(* IEC 61131-3 sources: std_i2980_v2.06_cp053/Source/IMM/ieccontrol/InjectionGeneral (part 8) *)

(* ---- ABInjectionCalibCycle.pu ---- *)
(*
@h    ! WARNING !
@h    The Kemro K2 system (including software) only meets category B according to EN 954-1,
@h    thus it is not intended for usage in safety-relevant control applications in the field
@h    of personal safety (e.g. emergency stop).
@h    To implement potentially necessary safety-relevant control tasks, always use additional
@h    external safety devices that are intended for the particular purpose, and meet the necessary
@h    functional safety.
@h    For further information see EN 954-1 (EN ISO 13849-1) and/or the K2-x00 user manual, chapter
@h    "CE conformity, directives and standards".

Do steps for automatic injection calibration (plant/dead time analysis)
*)

IMPORT_OVER_LISTFILE
 SET_EVENT
, SET_ALARM
, KMEM_ArrayCreate
, KMEM_ArraySet
, KMEM_ArrayDelete
, tnCalibMode_Both
, tnCalibState_Error
, tnCalibState_Aborted
, cMaxInjectionCount
, tnCalibMode_Raising
, tnCalibMode_Falling
, tnCalibState_Done
, cMoveFwd
, cMoveInject
, cMoveInjectCalib
, cMoveBwd
, cMoveDecompAftPlast
, nSetup
, tnCalibState_Running
, cCalibShiftData
, cCalibMeasuredVel
, cCalibMeasuredOutput
, tsControlParameters
, tnOperationMode
, tsDeviceId
, tsCalibMovement
, tsCalculatedInjectData2
, tsDeadTimeParameters
, tevStartRequest
, ABAutoCalibRedoListener
, tsCalculatedInjectData
, tevStartRequestData
, tyCalculatedDataArray
, tnCalibMode
, FBAutoCalibLog
, FBStopStartedMovements
, FBCheckReady
, tsCalibShiftData
, KMEM_CreateData
, KMEM_Status

END_IMPORT

ALGORITHM_BLOCK ABInjectionCalibCycle #DUMMY_EDIT_BLOCK

SYSTEM_VAR
 sv_bDoInjectionCalib : BOOL;
 sv_InjectControlParams : tsControlParameters;
 sv_OperationMode : tnOperationMode;
 sv_DeviceId : tsDeviceId;
 sv_CalibStateInjection : tsCalibMovement;
 sv_TmpInjectionData : tsCalculatedInjectData2;
 sv_InjectDeadTimeParams : tsDeadTimeParameters;
END_VAR

SYSTEM_OBJECT
 TaskMid : TASK;
 evStartRequest : tevStartRequest;
 PU_Task_7 : TASK;
END_OBJECT

VAR
 abAutoCalibRedoListenerInj : ABAutoCalibRedoListener;
END_VAR

PROCESS_ALGORITHM paRun ON TaskMid

VAR_TEMP
 tmpMeanData : tsCalculatedInjectData;
 i : DINT;
END_VAR

VAR
 evStartRequestData : tevStartRequestData;
 iInjectionCount : DINT;
 calculatedParameters : tyCalculatedDataArray;
 calibMode : tnCalibMode := tnCalibMode_Both;
 fbLog : FBAutoCalibLog;
 fbStopStartedMovements : FBStopStartedMovements;
 fbCheckReady : FBCheckReady;
 ShiftData : tsCalibShiftData;
 ShiftArrayCreateData : KMEM_CreateData;
 MeasuredVelArrayCreateData : KMEM_CreateData;
 MeasuredPosArrayCreateData : KMEM_CreateData;
 MeasuredOutputArrayCreateData : KMEM_CreateData;
 DifferencedArrayCreateData : KMEM_CreateData;
 SecondStageArrayCreateData : KMEM_CreateData;
 ThirdStageArrayCreateData : KMEM_CreateData;
 s : KMEM_Status;
 iSize : UDINT;
 rTmp : REAL;
END_VAR

(* IecGraph-Code *)

(* init step *)
INITIAL_STEP S_INIT:
AInit (P);
ACreateArrays (P);
END_STEP

ACTION AInit: #BEGIN_EDIT_BLOCK
sv_bDoInjectionCalib := TRUE;
iInjectionCount := 1;
sv_TmpInjectionData.CalibMode := calibMode;
sv_TmpInjectionData.bValid := FALSE;
sv_TmpInjectionData.bInvalid := FALSE;

;#END_EDIT_BLOCK END_ACTION (*AInit*)

(* steps *)
STEP S_RESET:
AStopmovements (P);
Action24 (P);
END_STEP

ACTION Action24: #BEGIN_EDIT_BLOCK
IF sv_CalibStateInjection.Status <> tnCalibState_Error THEN
   sv_CalibStateInjection.Status := tnCalibState_Aborted;
   fbLog('Injection calib aborted');
ELSE
    fbLog('Injection calib error');
END_IF;

;#END_EDIT_BLOCK END_ACTION (*Action24*)
STEP S_STOP:
ADeleteArrays (P);
Action22 (P);
END_STEP

ACTION Action22: #BEGIN_EDIT_BLOCK
sv_bDoInjectionCalib := FALSE;
STOP_PROCESS_ALGORITHM();

;#END_EDIT_BLOCK END_ACTION (*Action22*)
STEP S_DECOMP:
ADoDecompression (P);
Action8 (N);
END_STEP

ACTION Action8: #BEGIN_EDIT_BLOCK
fbCheckReady(DeviceId := sv_DeviceId)

;#END_EDIT_BLOCK END_ACTION (*Action8*)
STEP S_INJECT:
ADoProfile (P);
Action9 (N);
END_STEP

ACTION Action9: #BEGIN_EDIT_BLOCK
fbCheckReady(DeviceId := sv_DeviceId)

;#END_EDIT_BLOCK END_ACTION (*Action9*)
STEP S_WAIT_CALC:
END_STEP

STEP S_SAVE_CALC:
Action17 (P);
END_STEP

ACTION Action17: #BEGIN_EDIT_BLOCK
calculatedParameters[iInjectionCount] := sv_TmpInjectionData;

;#END_EDIT_BLOCK END_ACTION (*Action17*)
STEP S_NEXT_CYCLE:
Action16 (P);
END_STEP

ACTION Action16: #BEGIN_EDIT_BLOCK
iInjectionCount := iInjectionCount +1;

;#END_EDIT_BLOCK END_ACTION (*Action16*)
STEP S_DONE:
Action18 (P);
Action14 (P);
END_STEP

ACTION Action14: #BEGIN_EDIT_BLOCK
sv_CalibStateInjection.Status := tnCalibState_Done;

;#END_EDIT_BLOCK END_ACTION (*Action14*)

(* transitions *)
GO_ON_TRANSITION Trans15 (* Trans15 *) FROM S_RESET TO S_STOP :=  #BEGIN_EDIT_BLOCK
TRUE
;#END_EDIT_BLOCK
END_TRANSITION

TRANSITION Trans18 (* Trans18 *) FROM S_STOP TO S_INIT :=  #BEGIN_EDIT_BLOCK
TRUE
;#END_EDIT_BLOCK
END_TRANSITION

TRANSITION Trans1 (* Trans1 *) FROM S_INIT TO S_DECOMP :=  #BEGIN_EDIT_BLOCK
TRUE
;#END_EDIT_BLOCK
END_TRANSITION

TRANSITION Trans5 (* Trans5 *) FROM S_DECOMP TO S_INJECT :=  #BEGIN_EDIT_BLOCK
fbCheckReady.bReady
;#END_EDIT_BLOCK
END_TRANSITION

TRANSITION Trans2 (* Trans2 *) FROM S_INJECT TO S_WAIT_CALC :=  #BEGIN_EDIT_BLOCK
fbCheckReady.bReady
;#END_EDIT_BLOCK
END_TRANSITION

TRANSITION Trans21 (* Trans21 *) FROM S_WAIT_CALC TO S_SAVE_CALC :=  #BEGIN_EDIT_BLOCK
sv_TmpInjectionData.bValid
;#END_EDIT_BLOCK
END_TRANSITION

TRANSITION Trans22 (* Trans22 *) FROM S_WAIT_CALC TO S_RESET :=  #BEGIN_EDIT_BLOCK
sv_TmpInjectionData.bInvalid
;#END_EDIT_BLOCK
END_TRANSITION

TRANSITION Trans10 (* Trans10 *) FROM S_SAVE_CALC TO S_DONE :=  #BEGIN_EDIT_BLOCK
iInjectionCount >= cMaxInjectionCount
;#END_EDIT_BLOCK
END_TRANSITION

TRANSITION Trans11 (* Trans11 *) FROM S_SAVE_CALC TO S_NEXT_CYCLE :=  #BEGIN_EDIT_BLOCK
iInjectionCount < cMaxInjectionCount
;#END_EDIT_BLOCK
END_TRANSITION

TRANSITION Trans14 (* Trans14 *) FROM S_NEXT_CYCLE TO S_DECOMP :=  #BEGIN_EDIT_BLOCK
TRUE
;#END_EDIT_BLOCK
END_TRANSITION

TRANSITION Trans19 (* Trans19 *) FROM S_DONE TO S_STOP :=  #BEGIN_EDIT_BLOCK
TRUE
;#END_EDIT_BLOCK
END_TRANSITION

(* end IecGraph-Code *)
(* sfc-code *)

(* stand alone actions *)
ACTION ADoProfile: #BEGIN_EDIT_BLOCK
(**************************************** WARNING ********************************************
 *** The KEBA Kemro K2 System including software is not intended for safety control tasks! ***
 ***                       For further information see Comment tab!                        ***
 *********************************************************************************************)

evStartRequestData.DeviceId := sv_DeviceId;
evStartRequestData.MoveDir := cMoveFwd;
evStartRequestData.MoveId := cMoveInjectCalib;
SET_EVENT(evStartRequest, evStartRequestData);

;#END_EDIT_BLOCK END_ACTION (*ADoProfile*)
ACTION ADoDecompression: #BEGIN_EDIT_BLOCK
(**************************************** WARNING ********************************************
 *** The KEBA Kemro K2 System including software is not intended for safety control tasks! ***
 ***                       For further information see Comment tab!                        ***
 *********************************************************************************************)

evStartRequestData.DeviceId := sv_DeviceId;
evStartRequestData.MoveDir := cMoveBwd;
evStartRequestData.MoveId := cMoveDecompAftPlast;
SET_EVENT(evStartRequest, evStartRequestData);

;#END_EDIT_BLOCK END_ACTION (*ADoDecompression*)
ACTION AStopmovements: #BEGIN_EDIT_BLOCK
(**************************************** WARNING ********************************************
 *** The KEBA Kemro K2 System including software is not intended for safety control tasks! ***
 ***                       For further information see Comment tab!                        ***
 *********************************************************************************************)

fbStopStartedMovements();

;#END_EDIT_BLOCK END_ACTION (*AStopmovements*)
ACTION Action18: #BEGIN_EDIT_BLOCK
(**************************************** WARNING ********************************************
 *** The KEBA Kemro K2 System including software is not intended for safety control tasks! ***
 ***                       For further information see Comment tab!                        ***
 *********************************************************************************************)

tmpMeanData.rControllerKR := 0.0;
tmpMeanData.rControllerW  := 0.0;
tmpMeanData.tPlantDeadTime:= t#0ms;
tmpMeanData.rPlantK       := 0.0;
tmpMeanData.tPlantT1      := t#0ms;
tmpMeanData.tPlantT2      := t#0ms;
(* calculate mean value of all parameters *)
(* fixme: check if we need to calculate from falling and raising first
   and then calculate over the arry *)

FOR i:= 1 TO cMaxInjectionCount DO //FIXME: test
    IF calibMode = tnCalibMode_Both THEN
        tmpMeanData.rControllerKR := tmpMeanData.rControllerKR + calculatedParameters[i].Falling.rControllerKR + calculatedParameters[i].Raising.rControllerKR;
        tmpMeanData.rControllerW  := tmpMeanData.rControllerW  + calculatedParameters[i].Falling.rControllerW  + calculatedParameters[i].Raising.rControllerW;
        tmpMeanData.tPlantDeadTime:= tmpMeanData.tPlantDeadTime+ calculatedParameters[i].Falling.tPlantDeadTime+ calculatedParameters[i].Raising.tPlantDeadTime;
        tmpMeanData.rPlantK       := tmpMeanData.rPlantK       + calculatedParameters[i].Falling.rPlantK       + calculatedParameters[i].Raising.rPlantK;
        tmpMeanData.tPlantT1      := tmpMeanData.tPlantT1      + calculatedParameters[i].Falling.tPlantT1      + calculatedParameters[i].Raising.tPlantT1;
        tmpMeanData.tPlantT2      := tmpMeanData.tPlantT2      + calculatedParameters[i].Falling.tPlantT2      + calculatedParameters[i].Raising.tPlantT2;
    ELSIF calibMode = tnCalibMode_Raising THEN
        tmpMeanData.rControllerKR := tmpMeanData.rControllerKR + calculatedParameters[i].Raising.rControllerKR;
        tmpMeanData.rControllerW  := tmpMeanData.rControllerW  + calculatedParameters[i].Raising.rControllerW;
        tmpMeanData.tPlantDeadTime:= tmpMeanData.tPlantDeadTime+ calculatedParameters[i].Raising.tPlantDeadTime;
        tmpMeanData.rPlantK       := tmpMeanData.rPlantK       + calculatedParameters[i].Raising.rPlantK;
        tmpMeanData.tPlantT1      := tmpMeanData.tPlantT1      + calculatedParameters[i].Raising.tPlantT1;
        tmpMeanData.tPlantT2      := tmpMeanData.tPlantT2      + calculatedParameters[i].Raising.tPlantT2;
    ELSIF calibMode = tnCalibMode_Falling THEN
        tmpMeanData.rControllerKR := tmpMeanData.rControllerKR + calculatedParameters[i].Falling.rControllerKR ;
        tmpMeanData.rControllerW  := tmpMeanData.rControllerW  + calculatedParameters[i].Falling.rControllerW;
        tmpMeanData.tPlantDeadTime:= tmpMeanData.tPlantDeadTime+ calculatedParameters[i].Falling.tPlantDeadTime;
        tmpMeanData.rPlantK       := tmpMeanData.rPlantK       + calculatedParameters[i].Falling.rPlantK;
        tmpMeanData.tPlantT1      := tmpMeanData.tPlantT1      + calculatedParameters[i].Falling.tPlantT1;
        tmpMeanData.tPlantT2      := tmpMeanData.tPlantT2      + calculatedParameters[i].Falling.tPlantT2;
    END_IF;
END_FOR;

tmpMeanData.rControllerKR := tmpMeanData.rControllerKR / DINT_TO_REAL(cMaxInjectionCount);
tmpMeanData.rControllerW  := tmpMeanData.rControllerW  / DINT_TO_REAL(cMaxInjectionCount);
tmpMeanData.tPlantDeadTime:= tmpMeanData.tPlantDeadTime/ DINT_TO_REAL(cMaxInjectionCount);
tmpMeanData.rPlantK       := tmpMeanData.rPlantK       / DINT_TO_REAL(cMaxInjectionCount);
tmpMeanData.tPlantT1      := tmpMeanData.tPlantT1      / DINT_TO_REAL(cMaxInjectionCount);
tmpMeanData.tPlantT2      := tmpMeanData.tPlantT2      / DINT_TO_REAL(cMaxInjectionCount);

IF calibMode = tnCalibMode_Both THEN
    (* if only one edge no division is needed *)
    tmpMeanData.rControllerKR := tmpMeanData.rControllerKR / 2.0;
    tmpMeanData.rControllerW  := tmpMeanData.rControllerW  / 2.0;
    tmpMeanData.tPlantDeadTime:= DIVTIME(tmpMeanData.tPlantDeadTime, 2);
    tmpMeanData.rPlantK       := tmpMeanData.rPlantK/ 2.0;
    tmpMeanData.tPlantT1      := DIVTIME(tmpMeanData.tPlantT1, 2);
    tmpMeanData.tPlantT2      := DIVTIME(tmpMeanData.tPlantT2, 2);
END_IF;

sv_InjectDeadTimeParams.bCompensationEnabled := TRUE;
sv_InjectDeadTimeParams.dDeadTime := tmpMeanData.tPlantDeadTime;
sv_InjectDeadTimeParams.dPT2T1 := tmpMeanData.tPlantT1;
sv_InjectDeadTimeParams.dPT2T2 := tmpMeanData.tPlantT2;
sv_InjectDeadTimeParams.rPT2K  := tmpMeanData.rPlantK;

sv_InjectControlParams.rKS := 1.0;
sv_InjectControlParams.dTN := t#0s;
sv_InjectControlParams.dTV := t#0s;
sv_InjectControlParams.rP  := tmpMeanData.rControllerKR;

sv_InjectControlParams.bUsePIDControl := TRUE;

;#END_EDIT_BLOCK END_ACTION (*Action18*)
ACTION ACreateArrays: #BEGIN_EDIT_BLOCK
(**************************************** WARNING ********************************************
 *** The KEBA Kemro K2 System including software is not intended for safety control tasks! ***
 ***                       For further information see Comment tab!                        ***
 *********************************************************************************************)

//create dynamic arrays which are necessary for PID parameter detection
iSize := DINT_TO_UDINT(cMaxShiftData) + 1;
ShiftArrayCreateData := KMEM_ArrayCreate(cCalibShiftData, ShiftData, iSize);

iSize := DINT_TO_UDINT(cMaxRecordedData);
MeasuredVelArrayCreateData := KMEM_ArrayCreate(cCalibMeasuredVel, rTmp, iSize);
MeasuredPosArrayCreateData := KMEM_ArrayCreate(cCalibMeasuredPos, rTmp, iSize);
MeasuredOutputArrayCreateData := KMEM_ArrayCreate(cCalibMeasuredOutput, rTmp, iSize);

DifferencedArrayCreateData := KMEM_ArrayCreate(cCalibDifferenced, rTmp, iSize);
SecondStageArrayCreateData := KMEM_ArrayCreate(cCalibSecondStage, rTmp, iSize);
ThirdStageArrayCreateData := KMEM_ArrayCreate(cCalibThirdStage, rTmp, iSize);

;#END_EDIT_BLOCK END_ACTION (*ACreateArrays*)
ACTION ADeleteArrays: #BEGIN_EDIT_BLOCK
(**************************************** WARNING ********************************************
 *** The KEBA Kemro K2 System including software is not intended for safety control tasks! ***
 ***                       For further information see Comment tab!                        ***
 *********************************************************************************************)

s := KMEM_ArrayDelete(ShiftArrayCreateData.Handle);
s := KMEM_ArrayDelete(MeasuredVelArrayCreateData.Handle);
s := KMEM_ArrayDelete(MeasuredPosArrayCreateData.Handle);
s := KMEM_ArrayDelete(MeasuredOutputArrayCreateData.Handle);
s := KMEM_ArrayDelete(DifferencedArrayCreateData.Handle);
s := KMEM_ArrayDelete(SecondStageArrayCreateData.Handle);
s := KMEM_ArrayDelete(ThirdStageArrayCreateData.Handle);

;#END_EDIT_BLOCK END_ACTION (*ADeleteArrays*)

(* exits *)

EXIT_TRANSITION E_NotSetupMode := #BEGIN_EDIT_BLOCK
(**************************************** WARNING ********************************************
 *** The KEBA Kemro K2 System including software is not intended for safety control tasks! ***
 ***                       For further information see Comment tab!                        ***
 *********************************************************************************************)

sv_OperationMode <> nSetup
;#END_EDIT_BLOCK
PRIORITY 1 WITH  INITIAL_STEP S_RESET: END_STEP
END_TRANSITION

EXIT_TRANSITION E_NotCalibratingAnymore := #BEGIN_EDIT_BLOCK
// abort calibration, when not in running state and not finished
sv_CalibStateInjection.Status <> tnCalibState_Running AND (S_INIT.X OR S_DECOMP.X OR S_INJECT.X OR S_WAIT_CALC.X)
;#END_EDIT_BLOCK
PRIORITY 1 WITH  INITIAL_STEP S_RESET: END_STEP
END_TRANSITION
(* end sfc-code *)

END_ALGORITHM

POSTUPDATE_ALGORITHM pStart ON PU_Task_7 WITH sv_CalibStateInjection.Status

#BEGIN_EDIT_BLOCK
(**************************************** WARNING ********************************************
 *** The KEBA Kemro K2 System including software is not intended for safety control tasks! ***
 ***                       For further information see Comment tab!                        ***
 *********************************************************************************************)

IF sv_OperationMode = nSetup THEN
   IF sv_CalibStateInjection.Status = tnCalibState_Running THEN
      START_PROCESS_ALGORITHM(paRun);
   END_IF;
END_IF;

;#END_EDIT_BLOCK END_ALGORITHM

END_ALGORITHM_BLOCK

#END_OF_IEC_PART

@Puma @IecEditor 6 97 @Pou 25
@@@BEG_Comment@@@
@h    ! WARNING !
@h    The Kemro K2 system (including software) only meets category B according to EN 954-1,
@h    thus it is not intended for usage in safety-relevant control applications in the field
@h    of personal safety (e.g. emergency stop).
@h    To implement potentially necessary safety-relevant control tasks, always use additional
@h    external safety devices that are intended for the particular purpose, and meet the necessary
@h    functional safety.
@h    For further information see EN 954-1 (EN ISO 13849-1) and/or the K2-x00 user manual, chapter
@h    "CE conformity, directives and standards".

Do steps for automatic injection calibration (plant/dead time analysis)
@@@END_Comment@@@

@BEG_Contents

@BEG_Func
@RT(17)FuncTreeContainer
5
@Var @RT(9)SET_EVENT @RT(0) @T @T @DERIVED 0 @F @RT(23)KEBA_STANDARD_PROCEDURE @F
@T
@BEG_Attrib
0 @RT(0) @RT(0)
@END_Attrib
1 1 @F @F @F @F

@Var @RT(9)SET_ALARM @RT(0) @T @T @DERIVED 0 @F @RT(23)KEBA_STANDARD_PROCEDURE @F
@T
@BEG_Attrib
0 @RT(0) @RT(0)
@END_Attrib
1 1 @F @F @F @F

@Var @RT(16)KMEM_ArrayCreate @RT(0) @T @T @DERIVED 0 @F @RT(22)KEBA_STANDARD_FUNCTION @F
@T
@BEG_Attrib
0 @RT(0) @RT(0)
@END_Attrib
1 1 @F @F @F @F

@Var @RT(13)KMEM_ArraySet @RT(0) @T @T @DERIVED 0 @F @RT(22)KEBA_STANDARD_FUNCTION @F
@T
@BEG_Attrib
0 @RT(0) @RT(0)
@END_Attrib
1 1 @F @F @F @F

@Var @RT(16)KMEM_ArrayDelete @RT(0) @T @T @DERIVED 0 @F @RT(22)KEBA_STANDARD_FUNCTION @F
@T
@BEG_Attrib
0 @RT(0) @RT(0)
@END_Attrib
1 1 @F @F @F @F

@END_Func

@BEG_Const
@RT(18)ConstTreeContainer
17
@Var @RT(16)tnCalibMode_Both @RT(0) @T @T @DERIVED 0 @F @RT(11)tnCalibMode @F
@T
@BEG_Attrib
0 @RT(1)2 @RT(0)
@END_Attrib
1 1 @F @F @F @F

@Var @RT(18)tnCalibState_Error @RT(0) @T @T @DERIVED 0 @F @RT(12)tnCalibState @F
@T
@BEG_Attrib
0 @RT(1)3 @RT(32)error occured during calibration
@END_Attrib
1 1 @F @F @F @F

@Var @RT(20)tnCalibState_Aborted @RT(0) @T @T @DERIVED 0 @F @RT(12)tnCalibState @F
@T
@BEG_Attrib
0 @RT(1)4 @RT(19)calibration aborted
@END_Attrib
1 1 @F @F @F @F

@Var @RT(18)cMaxInjectionCount @RT(0) @T @F @DT @RT(4)DINT @RT(0) @T @T @BASIC 0 @F
@F @F
@T
@BEG_Attrib
0 @RT(1)3 @RT(41)how often to do injection for calibration
@END_Attrib
1 1 @F @F @F @F

@Var @RT(19)tnCalibMode_Raising @RT(0) @T @T @DERIVED 0 @F @RT(11)tnCalibMode @F
@T
@BEG_Attrib
0 @RT(1)0 @RT(0)
@END_Attrib
1 1 @F @F @F @F

@Var @RT(19)tnCalibMode_Falling @RT(0) @T @T @DERIVED 0 @F @RT(11)tnCalibMode @F
@T
@BEG_Attrib
0 @RT(1)1 @RT(0)
@END_Attrib
1 1 @F @F @F @F

@Var @RT(17)tnCalibState_Done @RT(0) @T @T @DERIVED 0 @F @RT(12)tnCalibState @F
@T
@BEG_Attrib
0 @RT(1)2 @RT(33)calibration finished successfully
@END_Attrib
1 1 @F @F @F @F

@Var @RT(8)cMoveFwd @RT(0) @T @F @DT @RT(4)DINT @RT(0) @T @T @BASIC 0 @F
@F @F
@T
@BEG_Attrib
0 @RT(2)12 @RT(16)movement forward
@END_Attrib
1 1 @F @F @F @F

@Var @RT(11)cMoveInject @RT(0) @T @F @DT @RT(4)DINT @RT(0) @T @T @BASIC 0 @F
@F @F
@T
@BEG_Attrib
0 @RT(2)14 @RT(15)inject movement
@END_Attrib
1 1 @F @F @F @F

@Var @RT(16)cMoveInjectCalib @RT(0) @T @F @DT @RT(4)DINT @RT(0) @T @T @BASIC 0 @F
@F @F
@T
@BEG_Attrib
0 @RT(2)70 @RT(48)calibration movement for servo inject controller
@END_Attrib
1 1 @F @F @F @F

@Var @RT(8)cMoveBwd @RT(0) @T @F @DT @RT(4)DINT @RT(0) @T @T @BASIC 0 @F
@F @F
@T
@BEG_Attrib
0 @RT(2)11 @RT(17)movement backward
@END_Attrib
1 1 @F @F @F @F

@Var @RT(19)cMoveDecompAftPlast @RT(0) @T @F @DT @RT(4)DINT @RT(0) @T @T @BASIC 0 @F
@F @F
@T
@BEG_Attrib
0 @RT(2)27 @RT(25)decompression after plast
@END_Attrib
1 1 @F @F @F @F

@Var @RT(6)nSetup @RT(0) @T @T @DERIVED 0 @F @RT(15)tnOperationMode @F
@T
@BEG_Attrib
0 @RT(1)0 @RT(36)Setup mode only for service engineer
@END_Attrib
1 1 @F @F @F @F

@Var @RT(20)tnCalibState_Running @RT(0) @T @T @DERIVED 0 @F @RT(12)tnCalibState @F
@T
@BEG_Attrib
0 @RT(1)1 @RT(23)calibration in progress
@END_Attrib
1 1 @F @F @F @F

@Var @RT(15)cCalibShiftData @RT(0) @T @F @DT @RT(10)STRING(31) @RT(0) @T @T @STRING 0 @F @RT(2)31 @F
@F @F
@T
@BEG_Attrib
0 @RT(11)'ShiftData' @RT(36)name of dynamic array for Shift Data
@END_Attrib
1 1 @F @F @F @F

@Var @RT(17)cCalibMeasuredVel @RT(0) @T @F @DT @RT(10)STRING(31) @RT(0) @T @T @STRING 0 @F @RT(2)31 @F
@F @F
@T
@BEG_Attrib
0 @RT(13)'MeasuredVel' @RT(97)name of dynamic array for measured velocities (used during automatic detection of PID parameters)
@END_Attrib
1 1 @F @F @F @F

@Var @RT(20)cCalibMeasuredOutput @RT(0) @T @F @DT @RT(10)STRING(31) @RT(0) @T @T @STRING 0 @F @RT(2)31 @F
@F @F
@T
@BEG_Attrib
0 @RT(16)'MeasuredOutput' @RT(100)name of dynamic array for measured output values (used during automatic detection of PID parameters)
@END_Attrib
1 1 @F @F @F @F

@END_Const

@BEG_Export

@BEG_Kind
@ALGORITHM_BLOCK @RT(21)ABInjectionCalibCycle @STRUCTURED_TEXT
@RT(0) @RT(0) @RT(0)
@END_Kind

@BEG_Dcl
@RT(16)DclTreeContainer
11
@Var @RT(20)sv_bDoInjectionCalib @RT(0) @T @F @DT @RT(4)BOOL @RT(0) @T @T @BASIC 0 @F
@F @F
@T
@BEG_Attrib
3 @RT(0) @RT(0) @RT(0)
@END_Attrib
1 8 @F @F @F @F

@Var @RT(22)sv_InjectControlParams @RT(0) @T @T @DERIVED 0 @T @T @DT @RT(19)tsControlParameters @RT(0) @T @T @UNKNOWN 0 @F
@F @F
@T
@BEG_Attrib
3 @RT(0) @RT(0) @RT(0)
@END_Attrib
1 8 @F @F @F @F

@Var @RT(16)sv_OperationMode @RT(0) @T @T @DERIVED 0 @T @T @DT @RT(15)tnOperationMode @RT(0) @T @T @UNKNOWN 0 @F
@F @F
@T
@BEG_Attrib
3 @RT(0) @RT(0) @RT(0)
@END_Attrib
1 8 @F @F @F @F

@Var @RT(11)sv_DeviceId @RT(0) @T @T @DERIVED 0 @T @T @DT @RT(10)tsDeviceId @RT(0) @T @T @UNKNOWN 0 @F
@F @F
@T
@BEG_Attrib
3 @RT(0) @RT(0) @RT(0)
@END_Attrib
1 8 @F @F @F @F

@Var @RT(22)sv_CalibStateInjection @RT(0) @T @T @DERIVED 0 @T @T @DT @RT(15)tsCalibMovement @RT(0) @T @T @UNKNOWN 0 @F
@F @F
@T
@BEG_Attrib
3 @RT(0) @RT(0) @RT(0)
@END_Attrib
1 8 @F @F @F @F

@Var @RT(19)sv_TmpInjectionData @RT(0) @T @T @DERIVED 0 @T @T @DT @RT(23)tsCalculatedInjectData2 @RT(0) @T @T @UNKNOWN 0 @F
@F @F
@T
@BEG_Attrib
3 @RT(0) @RT(0) @RT(0)
@END_Attrib
1 8 @F @F @F @F

@Var @RT(23)sv_InjectDeadTimeParams @RT(0) @T @T @DERIVED 0 @T @T @DT @RT(20)tsDeadTimeParameters @RT(0) @T @T @UNKNOWN 0 @F
@F @F
@T
@BEG_Attrib
3 @RT(0) @RT(0) @RT(0)
@END_Attrib
1 8 @F @F @F @F

@Var @RT(7)TaskMid @RT(0) @T @F @DT @RT(4)TASK @RT(0) @T @T @BASIC 0 @F
@F @F
@T
@BEG_Attrib
3 @RT(0) @RT(0) @RT(0)
@END_Attrib
1 7 @F @F @F @F

@Var @RT(14)evStartRequest @RT(0) @T @T @DERIVED 0 @T @T @DT @RT(15)tevStartRequest @RT(0) @T @T @UNKNOWN 0 @F
@F @F
@T
@BEG_Attrib
3 @RT(0) @RT(0) @RT(0)
@END_Attrib
1 7 @F @F @F @F

@Var @RT(9)PU_Task_7 @RT(0) @T @F @DT @RT(4)TASK @RT(0) @T @T @BASIC 0 @F
@F @F
@T
@BEG_Attrib
3 @RT(0) @RT(0) @RT(0)
@END_Attrib
1 7 @F @F @F @F

@Var @RT(26)abAutoCalibRedoListenerInj @RT(0) @T @T @DERIVED 0 @T @T @DT @RT(23)ABAutoCalibRedoListener @RT(0) @T @T @UNKNOWN 0 @F
@F @F
@T
@BEG_Attrib
3 @RT(0) @RT(0) @RT(0)
@END_Attrib
1 0 @F @F @F @F

@END_Dcl

@END_Export

@BEG_Body

2

@BEG_Export

@BEG_Algo
@PROCESS_ALGORITHM @RT(5)paRun @SEQUENTIAL_FLOW_CHART
@RT(0) @RT(0) @RT(7)TaskMid @F @F
@END_Algo

@BEG_Dcl
@RT(16)DclTreeContainer
20
@Var @RT(11)tmpMeanData @RT(0) @T @T @DERIVED 0 @T @T @DT @RT(22)tsCalculatedInjectData @RT(0) @T @T @UNKNOWN 0 @F
@F @F
@T
@BEG_Attrib
3 @RT(0) @RT(0) @RT(0)
@END_Attrib
1 4 @F @F @F @F

@Var @RT(1)i @RT(0) @T @F @DT @RT(4)DINT @RT(0) @T @T @BASIC 0 @F
@F @F
@T
@BEG_Attrib
3 @RT(0) @RT(0) @RT(0)
@END_Attrib
1 4 @F @F @F @F

@Var @RT(18)evStartRequestData @RT(0) @T @T @DERIVED 0 @T @T @DT @RT(19)tevStartRequestData @RT(0) @T @T @UNKNOWN 0 @F
@F @F
@T
@BEG_Attrib
3 @RT(0) @RT(0) @RT(0)
@END_Attrib
1 0 @F @F @F @F

@Var @RT(15)iInjectionCount @RT(0) @T @F @DT @RT(4)DINT @RT(0) @T @T @BASIC 0 @F
@F @F
@T
@BEG_Attrib
3 @RT(0) @RT(0) @RT(0)
@END_Attrib
1 0 @F @F @F @F

@Var @RT(20)calculatedParameters @RT(0) @T @T @DERIVED 0 @T @T @DT @RT(21)tyCalculatedDataArray @RT(0) @T @T @UNKNOWN 0 @F
@F @F
@T
@BEG_Attrib
3 @RT(0) @RT(0) @RT(0)
@END_Attrib
1 0 @F @F @F @F

@Var @RT(9)calibMode @RT(0) @T @T @DERIVED 0 @T @T @DT @RT(11)tnCalibMode @RT(0) @T @T @UNKNOWN 0 @F
@F @F
@T
@BEG_Attrib
3 @RT(16)tnCalibMode_Both @RT(0) @RT(0)
@END_Attrib
1 0 @F @F @F @F

@Var @RT(5)fbLog @RT(0) @T @T @DERIVED 0 @T @T @DT @RT(14)FBAutoCalibLog @RT(0) @T @T @UNKNOWN 0 @F
@F @F
@T
@BEG_Attrib
3 @RT(0) @RT(0) @RT(0)
@END_Attrib
1 0 @F @F @F @F

@Var @RT(22)fbStopStartedMovements @RT(0) @T @T @DERIVED 0 @T @T @DT @RT(22)FBStopStartedMovements @RT(0) @T @T @UNKNOWN 0 @F
@F @F
@T
@BEG_Attrib
3 @RT(0) @RT(0) @RT(0)
@END_Attrib
1 0 @F @F @F @F

@Var @RT(12)fbCheckReady @RT(0) @T @T @DERIVED 0 @T @T @DT @RT(12)FBCheckReady @RT(0) @T @T @UNKNOWN 0 @F
@F @F
@T
@BEG_Attrib
3 @RT(0) @RT(0) @RT(0)
@END_Attrib
1 0 @F @F @F @F

@Var @RT(9)ShiftData @RT(0) @T @T @DERIVED 0 @T @T @DT @RT(16)tsCalibShiftData @RT(0) @T @T @UNKNOWN 0 @F
@F @F
@T
@BEG_Attrib
3 @RT(0) @RT(0) @RT(0)
@END_Attrib
1 0 @F @F @F @F

@Var @RT(20)ShiftArrayCreateData @RT(0) @T @T @DERIVED 0 @T @T @DT @RT(15)KMEM_CreateData @RT(0) @T @T @UNKNOWN 0 @F
@F @F
@T
@BEG_Attrib
3 @RT(0) @RT(0) @RT(0)
@END_Attrib
1 0 @F @F @F @F

@Var @RT(26)MeasuredVelArrayCreateData @RT(0) @T @T @DERIVED 0 @T @T @DT @RT(15)KMEM_CreateData @RT(0) @T @T @UNKNOWN 0 @F
@F @F
@T
@BEG_Attrib
3 @RT(0) @RT(0) @RT(0)
@END_Attrib
1 0 @F @F @F @F

@Var @RT(26)MeasuredPosArrayCreateData @RT(0) @T @T @DERIVED 0 @T @T @DT @RT(15)KMEM_CreateData @RT(0) @T @T @UNKNOWN 0 @F
@F @F
@T
@BEG_Attrib
3 @RT(0) @RT(0) @RT(0)
@END_Attrib
1 0 @F @F @F @F

@Var @RT(29)MeasuredOutputArrayCreateData @RT(0) @T @T @DERIVED 0 @T @T @DT @RT(15)KMEM_CreateData @RT(0) @T @T @UNKNOWN 0 @F
@F @F
@T
@BEG_Attrib
3 @RT(0) @RT(0) @RT(0)
@END_Attrib
1 0 @F @F @F @F

@Var @RT(26)DifferencedArrayCreateData @RT(0) @T @T @DERIVED 0 @T @T @DT @RT(15)KMEM_CreateData @RT(0) @T @T @UNKNOWN 0 @F
@F @F
@T
@BEG_Attrib
3 @RT(0) @RT(0) @RT(0)
@END_Attrib
1 0 @F @F @F @F

@Var @RT(26)SecondStageArrayCreateData @RT(0) @T @T @DERIVED 0 @T @T @DT @RT(15)KMEM_CreateData @RT(0) @T @T @UNKNOWN 0 @F
@F @F
@T
@BEG_Attrib
3 @RT(0) @RT(0) @RT(0)
@END_Attrib
1 0 @F @F @F @F

@Var @RT(25)ThirdStageArrayCreateData @RT(0) @T @T @DERIVED 0 @T @T @DT @RT(15)KMEM_CreateData @RT(0) @T @T @UNKNOWN 0 @F
@F @F
@T
@BEG_Attrib
3 @RT(0) @RT(0) @RT(0)
@END_Attrib
1 0 @F @F @F @F

@Var @RT(1)s @RT(0) @T @T @DERIVED 0 @T @T @DT @RT(11)KMEM_Status @RT(0) @T @T @UNKNOWN 0 @F
@F @F
@T
@BEG_Attrib
3 @RT(0) @RT(0) @RT(0)
@END_Attrib
1 0 @F @F @F @F

@Var @RT(5)iSize @RT(0) @T @F @DT @RT(5)UDINT @RT(0) @T @T @BASIC 0 @F
@F @F
@T
@BEG_Attrib
3 @RT(0) @RT(0) @RT(0)
@END_Attrib
1 0 @F @F @F @F

@Var @RT(4)rTmp @RT(0) @T @F @DT @RT(4)REAL @RT(0) @T @T @BASIC 0 @F
@F @F
@T
@BEG_Attrib
3 @RT(0) @RT(0) @RT(0)
@END_Attrib
1 0 @F @F @F @F

@END_Dcl

@END_Export

@BEG_Export

@BEG_Algo
@POSTUPDATE_ALGORITHM @RT(6)pStart @STRUCTURED_TEXT
@RT(0) @RT(29)sv_CalibStateInjection.Status @RT(9)PU_Task_7 @F @F
@END_Algo

@BEG_Dcl
@RT(16)DclTreeContainer
0
@END_Dcl

@END_Export

@BEG_SfcBody
19 13 12

@BEG_SfcData 2
@StepSeq @RT(4)sseq @F 17
@Step @RT(7)S_RESET @F @F @T @F @RT(0) @F
@AcbCont @RT(7)unnamed @F 2
@Acb @RT(14)AStopmovements @F @F @RT(1)P @RT(0) @F @F @F @F
@Acb @RT(8)Action24 @F @T @RT(1)P @RT(0) @F @F @T @TL(7)
IF sv_CalibStateInjection.Status <> tnCalibState_Error THEN
   sv_CalibStateInjection.Status := tnCalibState_Aborted;
   fbLog('Injection calib aborted');
ELSE
    fbLog('Injection calib error');
END_IF;

@F

@Trans @RT(7)Trans15 @F @T @F @F @T @F @TL(2)
TRUE

@RT(7)Trans15 @F
@Step @RT(6)S_STOP @F @F @T @F @RT(0) @F
@AcbCont @RT(7)unnamed @F 2
@Acb @RT(13)ADeleteArrays @F @F @RT(1)P @RT(0) @F @F @F @F
@Acb @RT(8)Action22 @F @T @RT(1)P @RT(0) @F @F @T @TL(3)
sv_bDoInjectionCalib := FALSE;
STOP_PROCESS_ALGORITHM();

@F

@Trans @RT(7)Trans18 @F @T @F @F @T @T @TL(2)
TRUE

@RT(7)Trans18 @F
@Step @RT(6)S_INIT @F @T @F @F @RT(0) @F
@AcbCont @RT(7)unnamed @F 2
@Acb @RT(5)AInit @F @T @RT(1)P @RT(0) @F @F @T @TL(6)
sv_bDoInjectionCalib := TRUE;
iInjectionCount := 1;
sv_TmpInjectionData.CalibMode := calibMode;
sv_TmpInjectionData.bValid := FALSE;
sv_TmpInjectionData.bInvalid := FALSE;

@F
@Acb @RT(13)ACreateArrays @F @F @RT(1)P @RT(0) @F @F @F @F

@Trans @RT(6)Trans1 @F @T @F @F @T @T @TL(2)
TRUE

@RT(6)Trans1 @F
@Step @RT(8)S_DECOMP @F @F @T @F @RT(0) @F
@AcbCont @RT(7)unnamed @F 2
@Acb @RT(16)ADoDecompression @F @F @RT(1)P @RT(0) @F @F @F @F
@Acb @RT(7)Action8 @F @T @RT(1)N @RT(0) @F @F @T @TL(2)
fbCheckReady(DeviceId := sv_DeviceId)

@F

@Trans @RT(6)Trans5 @F @T @F @F @T @T @TL(2)
fbCheckReady.bReady

@RT(6)Trans5 @F
@Step @RT(8)S_INJECT @F @F @F @F @RT(0) @F
@AcbCont @RT(7)unnamed @F 2
@Acb @RT(10)ADoProfile @F @F @RT(1)P @RT(0) @F @F @F @F
@Acb @RT(7)Action9 @F @T @RT(1)N @RT(0) @F @F @T @TL(2)
fbCheckReady(DeviceId := sv_DeviceId)

@F

@Trans @RT(6)Trans2 @F @T @F @F @T @T @TL(2)
fbCheckReady.bReady

@RT(6)Trans2 @F
@Step @RT(11)S_WAIT_CALC @F @F @F @F @RT(0) @F
@AcbCont @RT(7)unnamed @F 0

@AltBranch @RT(3)alt @F 2
@TransSeq @RT(4)tseq @F 1
@Trans @RT(7)Trans21 @F @T @F @F @T @T @TL(2)
sv_TmpInjectionData.bValid

@RT(7)Trans21 @F

@TransSeq @RT(4)tseq @F 2
@Trans @RT(7)Trans22 @F @T @F @F @T @T @TL(2)
sv_TmpInjectionData.bInvalid

@RT(7)Trans22 @F
@Goto @RT(7)S_RESET @F @F

@Step @RT(11)S_SAVE_CALC @F @F @F @F @RT(0) @F
@AcbCont @RT(7)unnamed @F 1
@Acb @RT(8)Action17 @F @T @RT(1)P @RT(0) @F @F @T @TL(2)
calculatedParameters[iInjectionCount] := sv_TmpInjectionData;

@F

@AltBranch @RT(3)alt @F 2
@TransSeq @RT(4)tseq @F 1
@Trans @RT(7)Trans10 @F @T @F @F @T @T @TL(2)
iInjectionCount >= cMaxInjectionCount

@RT(7)Trans10 @F

@TransSeq @RT(4)tseq @F 4
@Trans @RT(7)Trans11 @F @T @F @F @T @T @TL(2)
iInjectionCount < cMaxInjectionCount

@RT(7)Trans11 @F
@Step @RT(12)S_NEXT_CYCLE @F @F @F @F @RT(0) @F
@AcbCont @RT(7)unnamed @F 1
@Acb @RT(8)Action16 @F @T @RT(1)P @RT(0) @F @F @T @TL(2)
iInjectionCount := iInjectionCount +1;

@F

@Trans @RT(7)Trans14 @F @T @F @F @T @T @TL(2)
TRUE

@RT(7)Trans14 @F
@Goto @RT(8)S_DECOMP @F @F

@Step @RT(6)S_DONE @F @F @F @F @RT(0) @F
@AcbCont @RT(7)unnamed @F 2
@Acb @RT(8)Action18 @F @F @RT(1)P @RT(0) @F @F @F @F
@Acb @RT(8)Action14 @F @T @RT(1)P @RT(0) @F @F @T @TL(2)
sv_CalibStateInjection.Status := tnCalibState_Done;

@F

@Trans @RT(7)Trans19 @F @T @F @F @T @T @TL(2)
TRUE

@RT(7)Trans19 @F
@Goto @RT(6)S_STOP @F @F
@END_SfcData
@SaActions 6
@SaText @RT(10)ADoProfile 1 @TL(10)
(**************************************** WARNING ********************************************
 *** The KEBA Kemro K2 System including software is not intended for safety control tasks! ***
 ***                       For further information see Comment tab!                        ***
 *********************************************************************************************)

evStartRequestData.DeviceId := sv_DeviceId;
evStartRequestData.MoveDir := cMoveFwd;
evStartRequestData.MoveId := cMoveInjectCalib;
SET_EVENT(evStartRequest, evStartRequestData);

@SaText @RT(16)ADoDecompression 1 @TL(10)
(**************************************** WARNING ********************************************
 *** The KEBA Kemro K2 System including software is not intended for safety control tasks! ***
 ***                       For further information see Comment tab!                        ***
 *********************************************************************************************)

evStartRequestData.DeviceId := sv_DeviceId;
evStartRequestData.MoveDir := cMoveBwd;
evStartRequestData.MoveId := cMoveDecompAftPlast;
SET_EVENT(evStartRequest, evStartRequestData);

@SaText @RT(14)AStopmovements 1 @TL(7)
(**************************************** WARNING ********************************************
 *** The KEBA Kemro K2 System including software is not intended for safety control tasks! ***
 ***                       For further information see Comment tab!                        ***
 *********************************************************************************************)

fbStopStartedMovements();

@SaText @RT(8)Action18 1 @TL(70)
(**************************************** WARNING ********************************************
 *** The KEBA Kemro K2 System including software is not intended for safety control tasks! ***
 ***                       For further information see Comment tab!                        ***
 *********************************************************************************************)

tmpMeanData.rControllerKR := 0.0;
tmpMeanData.rControllerW  := 0.0;
tmpMeanData.tPlantDeadTime:= t#0ms;
tmpMeanData.rPlantK       := 0.0;
tmpMeanData.tPlantT1      := t#0ms;
tmpMeanData.tPlantT2      := t#0ms;
(* calculate mean value of all parameters *)
(* fixme: check if we need to calculate from falling and raising first
   and then calculate over the arry *)

FOR i:= 1 TO cMaxInjectionCount DO //FIXME: test
    IF calibMode = tnCalibMode_Both THEN
        tmpMeanData.rControllerKR := tmpMeanData.rControllerKR + calculatedParameters[i].Falling.rControllerKR + calculatedParameters[i].Raising.rControllerKR;
        tmpMeanData.rControllerW  := tmpMeanData.rControllerW  + calculatedParameters[i].Falling.rControllerW  + calculatedParameters[i].Raising.rControllerW;
        tmpMeanData.tPlantDeadTime:= tmpMeanData.tPlantDeadTime+ calculatedParameters[i].Falling.tPlantDeadTime+ calculatedParameters[i].Raising.tPlantDeadTime;
        tmpMeanData.rPlantK       := tmpMeanData.rPlantK       + calculatedParameters[i].Falling.rPlantK       + calculatedParameters[i].Raising.rPlantK;
        tmpMeanData.tPlantT1      := tmpMeanData.tPlantT1      + calculatedParameters[i].Falling.tPlantT1      + calculatedParameters[i].Raising.tPlantT1;
        tmpMeanData.tPlantT2      := tmpMeanData.tPlantT2      + calculatedParameters[i].Falling.tPlantT2      + calculatedParameters[i].Raising.tPlantT2;
    ELSIF calibMode = tnCalibMode_Raising THEN
        tmpMeanData.rControllerKR := tmpMeanData.rControllerKR + calculatedParameters[i].Raising.rControllerKR;
        tmpMeanData.rControllerW  := tmpMeanData.rControllerW  + calculatedParameters[i].Raising.rControllerW;
        tmpMeanData.tPlantDeadTime:= tmpMeanData.tPlantDeadTime+ calculatedParameters[i].Raising.tPlantDeadTime;
        tmpMeanData.rPlantK       := tmpMeanData.rPlantK       + calculatedParameters[i].Raising.rPlantK;
        tmpMeanData.tPlantT1      := tmpMeanData.tPlantT1      + calculatedParameters[i].Raising.tPlantT1;
        tmpMeanData.tPlantT2      := tmpMeanData.tPlantT2      + calculatedParameters[i].Raising.tPlantT2;
    ELSIF calibMode = tnCalibMode_Falling THEN
        tmpMeanData.rControllerKR := tmpMeanData.rControllerKR + calculatedParameters[i].Falling.rControllerKR ;
        tmpMeanData.rControllerW  := tmpMeanData.rControllerW  + calculatedParameters[i].Falling.rControllerW;
        tmpMeanData.tPlantDeadTime:= tmpMeanData.tPlantDeadTime+ calculatedParameters[i].Falling.tPlantDeadTime;
        tmpMeanData.rPlantK       := tmpMeanData.rPlantK       + calculatedParameters[i].Falling.rPlantK;
        tmpMeanData.tPlantT1      := tmpMeanData.tPlantT1      + calculatedParameters[i].Falling.tPlantT1;
        tmpMeanData.tPlantT2      := tmpMeanData.tPlantT2      + calculatedParameters[i].Falling.tPlantT2;
    END_IF;
END_FOR;

tmpMeanData.rControllerKR := tmpMeanData.rControllerKR / DINT_TO_REAL(cMaxInjectionCount);
tmpMeanData.rControllerW  := tmpMeanData.rControllerW  / DINT_TO_REAL(cMaxInjectionCount);
tmpMeanData.tPlantDeadTime:= tmpMeanData.tPlantDeadTime/ DINT_TO_REAL(cMaxInjectionCount);
tmpMeanData.rPlantK       := tmpMeanData.rPlantK       / DINT_TO_REAL(cMaxInjectionCount);
tmpMeanData.tPlantT1      := tmpMeanData.tPlantT1      / DINT_TO_REAL(cMaxInjectionCount);
tmpMeanData.tPlantT2      := tmpMeanData.tPlantT2      / DINT_TO_REAL(cMaxInjectionCount);

IF calibMode = tnCalibMode_Both THEN
    (* if only one edge no division is needed *)
    tmpMeanData.rControllerKR := tmpMeanData.rControllerKR / 2.0;
    tmpMeanData.rControllerW  := tmpMeanData.rControllerW  / 2.0;
    tmpMeanData.tPlantDeadTime:= DIVTIME(tmpMeanData.tPlantDeadTime, 2);
    tmpMeanData.rPlantK       := tmpMeanData.rPlantK/ 2.0;
    tmpMeanData.tPlantT1      := DIVTIME(tmpMeanData.tPlantT1, 2);
    tmpMeanData.tPlantT2      := DIVTIME(tmpMeanData.tPlantT2, 2);
END_IF;

sv_InjectDeadTimeParams.bCompensationEnabled := TRUE;
sv_InjectDeadTimeParams.dDeadTime := tmpMeanData.tPlantDeadTime;
sv_InjectDeadTimeParams.dPT2T1 := tmpMeanData.tPlantT1;
sv_InjectDeadTimeParams.dPT2T2 := tmpMeanData.tPlantT2;
sv_InjectDeadTimeParams.rPT2K  := tmpMeanData.rPlantK;

sv_InjectControlParams.rKS := 1.0;
sv_InjectControlParams.dTN := t#0s;
sv_InjectControlParams.dTV := t#0s;
sv_InjectControlParams.rP  := tmpMeanData.rControllerKR;

sv_InjectControlParams.bUsePIDControl := TRUE;

@SaText @RT(13)ACreateArrays 1 @TL(18)
(**************************************** WARNING ********************************************
 *** The KEBA Kemro K2 System including software is not intended for safety control tasks! ***
 ***                       For further information see Comment tab!                        ***
 *********************************************************************************************)

//create dynamic arrays which are necessary for PID parameter detection
iSize := DINT_TO_UDINT(cMaxShiftData) + 1;
ShiftArrayCreateData := KMEM_ArrayCreate(cCalibShiftData, ShiftData, iSize);

iSize := DINT_TO_UDINT(cMaxRecordedData);
MeasuredVelArrayCreateData := KMEM_ArrayCreate(cCalibMeasuredVel, rTmp, iSize);
MeasuredPosArrayCreateData := KMEM_ArrayCreate(cCalibMeasuredPos, rTmp, iSize);
MeasuredOutputArrayCreateData := KMEM_ArrayCreate(cCalibMeasuredOutput, rTmp, iSize);

DifferencedArrayCreateData := KMEM_ArrayCreate(cCalibDifferenced, rTmp, iSize);
SecondStageArrayCreateData := KMEM_ArrayCreate(cCalibSecondStage, rTmp, iSize);
ThirdStageArrayCreateData := KMEM_ArrayCreate(cCalibThirdStage, rTmp, iSize);

@SaText @RT(13)ADeleteArrays 1 @TL(13)
(**************************************** WARNING ********************************************
 *** The KEBA Kemro K2 System including software is not intended for safety control tasks! ***
 ***                       For further information see Comment tab!                        ***
 *********************************************************************************************)

s := KMEM_ArrayDelete(ShiftArrayCreateData.Handle);
s := KMEM_ArrayDelete(MeasuredVelArrayCreateData.Handle);
s := KMEM_ArrayDelete(MeasuredPosArrayCreateData.Handle);
s := KMEM_ArrayDelete(MeasuredOutputArrayCreateData.Handle);
s := KMEM_ArrayDelete(DifferencedArrayCreateData.Handle);
s := KMEM_ArrayDelete(SecondStageArrayCreateData.Handle);
s := KMEM_ArrayDelete(ThirdStageArrayCreateData.Handle);

@SaTrans 0
@SaExits 2
@SaExit @SaText @RT(14)E_NotSetupMode 1 @TL(7)
(**************************************** WARNING ********************************************
 *** The KEBA Kemro K2 System including software is not intended for safety control tasks! ***
 ***                       For further information see Comment tab!                        ***
 *********************************************************************************************)

sv_OperationMode <> nSetup

@RT(7)S_RESET @RT(1)1 @F @F @SaSfc @RT(14)E_NotSetupMode 5 @RT(5)DUMMY
@BEG_SfcData 2
@ExitSeq @RT(4)sseq @F 3
@Step @RT(8)unnamed1 @F @T @F @F @RT(0) @F
@AcbCont @RT(7)unnamed @F 0

@Trans @RT(8)unnamed3 @F @T @F @F @T @T @TL(2)

@RT(8)unnamed3 @F
@Goto @RT(9)unlabeled @F @F
@END_SfcData

@SaExit @SaText @RT(23)E_NotCalibratingAnymore 1 @TL(3)
// abort calibration, when not in running state and not finished
sv_CalibStateInjection.Status <> tnCalibState_Running AND (S_INIT.X OR S_DECOMP.X OR S_INJECT.X OR S_WAIT_CALC.X)

@RT(7)S_RESET @RT(1)1 @F @F @SaSfc @RT(23)E_NotCalibratingAnymore 5 @RT(5)DUMMY
@BEG_SfcData 2
@ExitSeq @RT(4)sseq @F 3
@Step @RT(8)unnamed4 @F @T @F @F @RT(0) @F
@AcbCont @RT(7)unnamed @F 0

@Trans @RT(8)unnamed6 @F @T @F @F @T @T @TL(2)

@RT(8)unnamed6 @F
@Goto @RT(9)unlabeled @F @F
@END_SfcData

@END_SfcBody

@@@BEG_Comment@@@
@TL(0)

@@@END_Comment@@@

@BEG_Body
@TL(12)
(**************************************** WARNING ********************************************
 *** The KEBA Kemro K2 System including software is not intended for safety control tasks! ***
 ***                       For further information see Comment tab!                        ***
 *********************************************************************************************)

IF sv_OperationMode = nSetup THEN
   IF sv_CalibStateInjection.Status = tnCalibState_Running THEN
      START_PROCESS_ALGORITHM(paRun);
   END_IF;
END_IF;

@END_Body

@@@BEG_Comment@@@
@TL(0)

@@@END_Comment@@@
@END_Body

@END_Contents

(* ---- ABManualButton.pu ---- *)
IMPORT_OVER_LISTFILE
 cMoveFwd
, cMoveBwd
, cMovePlast
, cCompAutoPurge
, FBManualButton
, FBManualButtonKeep
, tsDeviceId
, tnOperationMode
, FBCheckReady

END_IMPORT

ALGORITHM_BLOCK ABManualButton #DUMMY_EDIT_BLOCK

SYSTEM_VAR
 sv_bInitDone : BOOL;
 sv_DeviceId : tsDeviceId;
 sv_OperationMode : tnOperationMode;
END_VAR

SYSTEM_OBJECT
 PU_Task_7 : TASK;
END_OBJECT

VAR
 fbManualButton : FBManualButton;
 fbManualButtonPlast : FBManualButtonKeep;
 mpbAutoPurgeReady : REFTO BOOL;
END_VAR

ALGORITHM aButtonInject

VAR_INPUT
 bButtonInject : BOOL;
END_VAR
#BEGIN_EDIT_BLOCK
(**************************************** WARNING ********************************************
 *** The KEBA Kemro K2 System including software is not intended for safety control tasks! ***
 ***                       For further information see Comment tab!                        ***
 *********************************************************************************************)

IF mpbAutoPurgeReady <> EMPTY AND NOT mpbAutoPurgeReady^ THEN
    // autopurge available and active -> ignore manual button
    RETURN;
END_IF;

fbManualButton(bButton := bButtonInject, MoveId := cMoveInject, MoveDir :=cMoveFwd);

;#END_EDIT_BLOCK END_ALGORITHM

ALGORITHM aButtonDecomp

VAR_INPUT
 bButtonDecomp : BOOL;
END_VAR
#BEGIN_EDIT_BLOCK
(**************************************** WARNING ********************************************
 *** The KEBA Kemro K2 System including software is not intended for safety control tasks! ***
 ***                       For further information see Comment tab!                        ***
 *********************************************************************************************)

IF mpbAutoPurgeReady <> EMPTY AND NOT mpbAutoPurgeReady^ THEN
    // autopurge available and active -> ignore manual button
    RETURN;
END_IF;

fbManualButton(bButton := bButtonDecomp, MoveId := cMoveDecompAftPlast, MoveDir := cMoveBwd);

;#END_EDIT_BLOCK END_ALGORITHM

ALGORITHM aButtonPlast

VAR_INPUT
 bButtonPlast : BOOL;
END_VAR
#BEGIN_EDIT_BLOCK
(**************************************** WARNING ********************************************
 *** The KEBA Kemro K2 System including software is not intended for safety control tasks! ***
 ***                       For further information see Comment tab!                        ***
 *********************************************************************************************)

IF mpbAutoPurgeReady <> EMPTY AND NOT mpbAutoPurgeReady^ THEN
    // autopurge available and active -> ignore manual button
    RETURN;
END_IF;

IF sv_OperationMode = nManual THEN
   //plast in manual mode should also contain decomp before and decomp after
   //-> send start request for combined plast movement
   fbManualButtonPlast(bButton := bButtonPlast, MoveId := cMoveCombinedPlast, MoveDir := cMoveBwd);
ELSE
   //in setup mode only plast should be executed
   fbManualButtonPlast(bButton := bButtonPlast, MoveId := cMovePlast, MoveDir := cMoveBwd);
END_IF;

;#END_EDIT_BLOCK END_ALGORITHM

POSTUPDATE_ALGORITHM pInitDone ON PU_Task_7(10) WITH sv_bInitDone

VAR
 fbCheckAutoPurgeReady : FBCheckReady;
 DeviceIdAutoPurge : tsDeviceId;
END_VAR
#BEGIN_EDIT_BLOCK
(**************************************** WARNING ********************************************
 *** The KEBA Kemro K2 System including software is not intended for safety control tasks! ***
 ***                       For further information see Comment tab!                        ***
 *********************************************************************************************)

//get reference to ready flag of autopurge movement
DeviceIdAutoPurge.CompId := cCompAutoPurge;
DeviceIdAutoPurge.IndexId := sv_DeviceId.IndexId;

fbCheckAutoPurgeReady(DeviceId := DeviceIdAutoPurge);
mpbAutoPurgeReady := fbCheckAutoPurgeReady.pbReady;

;#END_EDIT_BLOCK END_ALGORITHM

END_ALGORITHM_BLOCK

#END_OF_IEC_PART

@Puma @IecEditor 6 30 @Pou 25
@@@BEG_Comment@@@

@@@END_Comment@@@

@BEG_Contents

@BEG_Func
@RT(17)FuncTreeContainer
0
@END_Func

@BEG_Const
@RT(18)ConstTreeContainer
4
@Var @RT(8)cMoveFwd @RT(0) @T @F @DT @RT(4)DINT @RT(0) @T @T @BASIC 0 @F
@F @F
@T
@BEG_Attrib
0 @RT(2)12 @RT(16)movement forward
@END_Attrib
1 1 @F @F @F @F

@Var @RT(8)cMoveBwd @RT(0) @T @F @DT @RT(4)DINT @RT(0) @T @T @BASIC 0 @F
@F @F
@T
@BEG_Attrib
0 @RT(2)11 @RT(17)movement backward
@END_Attrib
1 1 @F @F @F @F

@Var @RT(10)cMovePlast @RT(0) @T @F @DT @RT(4)DINT @RT(0) @T @T @BASIC 0 @F
@F @F
@T
@BEG_Attrib
0 @RT(2)13 @RT(23)plast movement (rotate)
@END_Attrib
1 1 @F @F @F @F

@Var @RT(14)cCompAutoPurge @RT(0) @T @F @DT @RT(4)DINT @RT(0) @T @T @BASIC 0 @F
@F @F
@T
@BEG_Attrib
0 @RT(3)126 @RT(19)Component AutoPurge
@END_Attrib
1 1 @F @F @F @F

@END_Const

@BEG_Export

@BEG_Kind
@ALGORITHM_BLOCK @RT(14)ABManualButton @STRUCTURED_TEXT
@RT(0) @RT(0) @RT(0)
@END_Kind

@BEG_Dcl
@RT(16)DclTreeContainer
7
@Var @RT(9)PU_Task_7 @RT(0) @T @T @RENAMED 0 @T @T @DT @RT(4)TASK @RT(0) @T @T @BASIC 0 @F
@F @F
@T
@BEG_Attrib
3 @RT(0) @RT(0) @RT(0)
@END_Attrib
1 7 @F @F @F @F

@Var @RT(14)fbManualButton @RT(0) @T @T @DERIVED 0 @T @T @DT @RT(14)FBManualButton @RT(0) @T @T @UNKNOWN 0 @F
@F @F
@T
@BEG_Attrib
3 @RT(0) @RT(0) @RT(0)
@END_Attrib
1 0 @F @F @F @F

@Var @RT(19)fbManualButtonPlast @RT(0) @T @T @DERIVED 0 @T @T @DT @RT(18)FBManualButtonKeep @RT(0) @T @T @UNKNOWN 0 @F
@F @F
@T
@BEG_Attrib
3 @RT(0) @RT(0) @RT(0)
@END_Attrib
1 0 @F @F @F @F

@Var @RT(12)sv_bInitDone @RT(0) @T @T @RENAMED 0 @T @T @DT @RT(4)BOOL @RT(0) @T @T @BASIC 0 @F
@F @F
@T
@BEG_Attrib
3 @RT(0) @RT(0) @RT(0)
@END_Attrib
1 8 @F @F @F @F

@Var @RT(11)sv_DeviceId @RT(0) @T @T @DERIVED 0 @T @T @DT @RT(10)tsDeviceId @RT(0) @T @T @UNKNOWN 0 @F
@F @F
@T
@BEG_Attrib
3 @RT(0) @RT(0) @RT(0)
@END_Attrib
1 8 @F @F @F @F

@Var @RT(16)sv_OperationMode @RT(0) @T @T @RENAMED 0 @T @T @DT @RT(15)tnOperationMode @RT(0) @T @T @UNKNOWN 0 @F
@F @F
@T
@BEG_Attrib
3 @RT(0) @RT(0) @RT(0)
@END_Attrib
1 8 @F @F @F @F

@Var @RT(17)mpbAutoPurgeReady @RT(0) @T @T @REFTO 0 @T @DT @RT(4)BOOL @RT(0) @T @T @BASIC 0 @F
@F @F
@T
@BEG_Attrib
3 @RT(0) @RT(0) @RT(0)
@END_Attrib
1 0 @F @F @F @F

@END_Dcl

@END_Export

@BEG_Body

4

@BEG_Export

@BEG_Algo
@ALGORITHM @RT(13)aButtonInject @STRUCTURED_TEXT
@RT(0) @RT(0) @RT(0) @F @F
@END_Algo

@BEG_Dcl
@RT(16)DclTreeContainer
1
@Var @RT(13)bButtonInject @RT(0) @T @F @DT @RT(4)BOOL @RT(0) @T @T @BASIC 0 @F
@F @F
@T
@BEG_Attrib
3 @RT(0) @RT(0) @RT(0)
@END_Attrib
1 1 @F @F @F @F

@END_Dcl

@END_Export

@BEG_Export

@BEG_Algo
@ALGORITHM @RT(13)aButtonDecomp @STRUCTURED_TEXT
@RT(0) @RT(0) @RT(0) @F @F
@END_Algo

@BEG_Dcl
@RT(16)DclTreeContainer
1
@Var @RT(13)bButtonDecomp @RT(0) @T @F @DT @RT(4)BOOL @RT(0) @T @T @BASIC 0 @F
@F @F
@T
@BEG_Attrib
3 @RT(0) @RT(0) @RT(0)
@END_Attrib
1 1 @F @F @F @F

@END_Dcl

@END_Export

@BEG_Export

@BEG_Algo
@ALGORITHM @RT(12)aButtonPlast @STRUCTURED_TEXT
@RT(0) @RT(0) @RT(0) @F @F
@END_Algo

@BEG_Dcl
@RT(16)DclTreeContainer
1
@Var @RT(12)bButtonPlast @RT(0) @T @F @DT @RT(4)BOOL @RT(0) @T @T @BASIC 0 @F
@F @F
@T
@BEG_Attrib
3 @RT(0) @RT(0) @RT(0)
@END_Attrib
1 1 @F @F @F @F

@END_Dcl

@END_Export

@BEG_Export

@BEG_Algo
@POSTUPDATE_ALGORITHM @RT(9)pInitDone @STRUCTURED_TEXT
@RT(0) @RT(12)sv_bInitDone @RT(13)PU_Task_7(10) @F @F
@END_Algo

@BEG_Dcl
@RT(16)DclTreeContainer
2
@Var @RT(21)fbCheckAutoPurgeReady @RT(0) @T @T @DERIVED 0 @T @T @DT @RT(12)FBCheckReady @RT(0) @T @T @UNKNOWN 0 @F
@F @F
@T
@BEG_Attrib
3 @RT(0) @RT(0) @RT(0)
@END_Attrib
1 0 @F @F @F @F

@Var @RT(17)DeviceIdAutoPurge @RT(0) @T @T @DERIVED 0 @T @T @DT @RT(10)tsDeviceId @RT(0) @T @T @UNKNOWN 0 @F
@F @F
@T
@BEG_Attrib
3 @RT(0) @RT(0) @RT(0)
@END_Attrib
1 0 @F @F @F @F

@END_Dcl

@END_Export

@BEG_Body
@TL(12)
(**************************************** WARNING ********************************************
 *** The KEBA Kemro K2 System including software is not intended for safety control tasks! ***
 ***                       For further information see Comment tab!                        ***
 *********************************************************************************************)

IF mpbAutoPurgeReady <> EMPTY AND NOT mpbAutoPurgeReady^ THEN
    // autopurge available and active -> ignore manual button
    RETURN;
END_IF;

fbManualButton(bButton := bButtonInject, MoveId := cMoveInject, MoveDir :=cMoveFwd);

@END_Body

@@@BEG_Comment@@@
@TL(0)

@@@END_Comment@@@

@BEG_Body
@TL(13)
(**************************************** WARNING ********************************************
 *** The KEBA Kemro K2 System including software is not intended for safety control tasks! ***
 ***                       For further information see Comment tab!                        ***
 *********************************************************************************************)

IF mpbAutoPurgeReady <> EMPTY AND NOT mpbAutoPurgeReady^ THEN
    // autopurge available and active -> ignore manual button
    RETURN;
END_IF;

fbManualButton(bButton := bButtonDecomp, MoveId := cMoveDecompAftPlast, MoveDir := cMoveBwd);

@END_Body

@@@BEG_Comment@@@
@TL(0)

@@@END_Comment@@@

@BEG_Body
@TL(20)
(**************************************** WARNING ********************************************
 *** The KEBA Kemro K2 System including software is not intended for safety control tasks! ***
 ***                       For further information see Comment tab!                        ***
 *********************************************************************************************)

IF mpbAutoPurgeReady <> EMPTY AND NOT mpbAutoPurgeReady^ THEN
    // autopurge available and active -> ignore manual button
    RETURN;
END_IF;

IF sv_OperationMode = nManual THEN
   //plast in manual mode should also contain decomp before and decomp after
   //-> send start request for combined plast movement
   fbManualButtonPlast(bButton := bButtonPlast, MoveId := cMoveCombinedPlast, MoveDir := cMoveBwd);
ELSE
   //in setup mode only plast should be executed
   fbManualButtonPlast(bButton := bButtonPlast, MoveId := cMovePlast, MoveDir := cMoveBwd);
END_IF;

@END_Body

@@@BEG_Comment@@@
@TL(0)

@@@END_Comment@@@

@BEG_Body
@TL(14)
(**************************************** WARNING ********************************************
 *** The KEBA Kemro K2 System including software is not intended for safety control tasks! ***
 ***                       For further information see Comment tab!                        ***
 *********************************************************************************************)

//get reference to ready flag of autopurge movement
DeviceIdAutoPurge.CompId := cCompAutoPurge;
DeviceIdAutoPurge.IndexId := sv_DeviceId.IndexId;

fbCheckAutoPurgeReady(DeviceId := DeviceIdAutoPurge);
mpbAutoPurgeReady := fbCheckAutoPurgeReady.pbReady;

@END_Body

@@@BEG_Comment@@@
@TL(0)

@@@END_Comment@@@
@END_Body

@END_Contents

(* ---- ABMoveCombinedPlast.pu ---- *)
(*
@h    ! WARNING !
@h    The Kemro K2 system (including software) only meets category B according to EN 954-1,
@h    thus it is not intended for usage in safety-relevant control applications in the field
@h    of personal safety (e.g. emergency stop).
@h    To implement potentially necessary safety-relevant control tasks, always use additional
@h    external safety devices that are intended for the particular purpose, and meet the necessary
@h    functional safety.
@h    For further information see EN 954-1 (EN ISO 13849-1) and/or the K2-x00 user manual, chapter
@h    "CE conformity, directives and standards".

ABMoveCombinedPlast is a combination of the following movements:
- decompression before plast
- plast
- decompression after plast

Therefore the movement sv_MoveCombinedPlast is registered

After receiving a start event for the movement with moveId cMoveCombinedPlast this block
coordinates decompression and plast by sending the start events to this movements.

Attention:
To avoid that autocycle continues to early the pbDeviceReady flag is modified.
During this combined movement is active, pbDeviceReady refers to sv_bCombinedPlastReady.
After the movement was stopped or it is finished, pbDeviceReady refers to sv_bDeviceReady again.
*)

IMPORT_OVER_LISTFILE
 SET_EVENT
, cCompInjection
, cMoveDecompBefPlast
, cMoveCombinedPlast
, tsMoveData
, tevStart
, tevStop
, tsDeviceId
, FBDebugTrace
, tsTraceLevel
, tDeviceMovementList
, tevStartedStopped
, tevStartedStoppedData
, tsCombinedPlastData
, KAPPL_VisProfilePlast
, tsSetTimes
, tsDecompParam
, tnOperationMode
, tsActTimes
, ABMovementRegister
, tevStartData
, tevStopData
, FBStart
, FBDebugTrace2
, TON
, FBUpdateEditorProperties

END_IMPORT

ALGORITHM_BLOCK ABMoveCombinedPlast #DUMMY_EDIT_BLOCK

SYSTEM_VAR
 sv_MoveCombinedPlast : tsMoveData (* combined plast movement (decomp bef -> plast -> decomp after) *);
 sv_bInitStart : BOOL;
 sv_DeviceId : tsDeviceId;
 sv_TraceLevel : tsTraceLevel;
 sv_bDeviceReady : BOOL;
 sv_DeviceMovements : tDeviceMovementList;
 sv_bCombinedPlastReady : BOOL (* combined plast ready *);
 sv_CombinedPlastData : tsCombinedPlastData (* necessary data for diplaying combined plast movement in odc editor *);
 sv_PlastProfVis : KAPPL_VisProfilePlast;
 sv_dCalculatedDurationDecompAft : TIME;
 sv_dCalculatedDurationDecompBef : TIME;
 sv_dCalculatedDurationPlast : TIME;
 sv_dDurationCombinedPlast : TIME (* Calculated duration for combined plasticizing *);
 sv_PlastTimesSet : tsSetTimes;
 sv_DecompAftPlastSettings : tsDecompParam;
 sv_DecompBefPlastSettings : tsDecompParam;
 sv_DecompTimesSet : tsSetTimes;
 sv_bPlastEndReached : BOOL (* flag if plast icizing endposition is reached *);
 sv_OperationMode : tnOperationMode;
 sv_rTargetValueDecBefPlast : REAL (* target value of decomp before plast (in cmł) *);
 sv_dActPlastDecompTime : TIME (* act time for combined plast movement *);
 sv_bActivatedDecompBeforePlast : BOOL (* indicates if movement decompress should be activated if start event is sent *);
 sv_bActivatedDecompAfterPlast : BOOL (* indicates if movement decompress should be activated if start event is sent *);
 sv_bMoveRegisterDone : BOOL;
 sv_PlastTimesAct : tsActTimes;
 sv_rPlastStartPosition : REAL (* position at starting plasticizing *);
 sv_rPlastEndPosition : REAL (* position at end of plasticizing *);
 sv_rScrewPosition : REAL (* specific screw position im cmł *);
END_VAR

SYSTEM_OBJECT
 PU_Task_7 : TASK;
 EV_Task_3 : TASK;
 evStart : tevStart;
 evStop : tevStop;
 evStartedStopped : tevStartedStopped;
 TaskSequencer : TASK;
END_OBJECT

VAR
 mbStop : BOOL;
 fbDebugTrace : FBDebugTrace;
 evStartedStoppedData : tevStartedStoppedData;
 miIndex : DINT (* index of this FU in sv_DeviceMovement - list *);
END_VAR

ALGORITHM aRegister

VAR
 abCombinedPlastRegister : ABMovementRegister;
END_VAR
#BEGIN_EDIT_BLOCK
(**************************************** WARNING ********************************************
 *** The KEBA Kemro K2 System including software is not intended for safety control tasks! ***
 ***                       For further information see Comment tab!                        ***
 *********************************************************************************************)

//register inject movement
sv_MoveCombinedPlast.LockGroups[1] := cLockGroupHeatingNozzle;
sv_MoveCombinedPlast.LockGroups[2] := cLockGroupSafetyGateNozzle;
sv_MoveCombinedPlast.LockGroups[3] := cLockGroupSafetyGateMold;
sv_MoveCombinedPlast.sIconPath := CONCAT(GET_MY_FU_NAME(),"\hmi\images\movScrewRotate.gif");

abCombinedPlastRegister.aRegister(@sv_MoveCombinedPlast);

;#END_EDIT_BLOCK END_ALGORITHM

POSTUPDATE_ALGORITHM pInitStart ON PU_Task_7 WITH sv_bInitStart

#BEGIN_EDIT_BLOCK
(**************************************** WARNING ********************************************
 *** The KEBA Kemro K2 System including software is not intended for safety control tasks! ***
 ***                       For further information see Comment tab!                        ***
 *********************************************************************************************)

IF sv_bInitStart THEN
   aRegister();
END_IF;

;#END_EDIT_BLOCK END_ALGORITHM

(*
This Algo receives the evStart event, checks the startconditions and starts paMoveControl.

*)

EVENT_ALGORITHM evaStart ON EV_Task_3 WITH evStart

VAR_INPUT
 evStartData : tevStartData;
END_VAR
#BEGIN_EDIT_BLOCK
(**************************************** WARNING ********************************************
 *** The KEBA Kemro K2 System including software is not intended for safety control tasks! ***
 ***                       For further information see Comment tab!                        ***
 *********************************************************************************************)

IF evStartData.DeviceId.CompId = sv_DeviceId.CompId AND
   evStartData.DeviceId.IndexId = sv_DeviceId.IndexId  THEN

   IF evStartData.MoveId = cMoveCombinedPlast THEN

      //modify pbDeviceReady
      sv_DeviceMovements[miIndex].pbDeviceReady := @sv_bCombinedPlastReady;

      // sending stopped-Message
      evStartedStoppedData.DeviceId := sv_DeviceId;
      evStartedStoppedData.MoveId := cMoveCombinedPlast;
      evStartedStoppedData.MoveDir := cMoveBwd;
      evStartedStoppedData.State := nStarted;
      SET_EVENT(evStartedStopped,evStartedStoppedData);

      sv_bCombinedPlastReady := FALSE;
      mbStop := FALSE;

      START_PROCESS_ALGORITHM(paMoveControl);
   END_IF;

END_IF;

;#END_EDIT_BLOCK END_ALGORITHM

(*
Receives the stopevent and signalls paMoveControl to stop the running movement.
*)

EVENT_ALGORITHM evaStop ON EV_Task_3 WITH evStop

VAR_INPUT
 evStopData : tevStopData;
END_VAR
#BEGIN_EDIT_BLOCK
(**************************************** WARNING ********************************************
 *** The KEBA Kemro K2 System including software is not intended for safety control tasks! ***
 ***                       For further information see Comment tab!                        ***
 *********************************************************************************************)

IF evStopData.DeviceId = sv_DeviceId THEN

    IF sv_TraceLevel.bDeviceState THEN
            fbDebugTrace(sText := 'ABMoveCombinedPlast : evStop received');
    END_IF;

   //stopping movement
   mbStop := TRUE;
END_IF;

;#END_EDIT_BLOCK END_ALGORITHM

PROCESS_ALGORITHM paMoveControl ON TaskSequencer(1)

VAR_TEMP
 b : BOOL;
END_VAR

VAR
 fbStart : FBStart;
 fbDebugTrace2 : FBDebugTrace2;
 fbMoveTime : TON;
 dNull : TIME;
END_VAR

(* IecGraph-Code *)

(* init step *)
INITIAL_STEP S_Init:
END_STEP

(* steps *)
STEP S_Start:
AStart (P);
AMoveTime (S);
END_STEP

ACTION AStart: #BEGIN_EDIT_BLOCK
fbDebugTrace2(nDeviceState, 'Combined Plast Started');
fbMoveTime(IN := FALSE,
           PT := t#20d);

;#END_EDIT_BLOCK END_ACTION (*AStart*)
STEP S_DecBefPlast:
AStartDecBefPlast (P);
END_STEP

ACTION AStartDecBefPlast: #BEGIN_EDIT_BLOCK
fbStart(DeviceId := sv_DeviceId,
        MoveDir := cMoveBwd,
        MoveId := cMoveDecompBefPlast);

;#END_EDIT_BLOCK END_ACTION (*AStartDecBefPlast*)
STEP S_Plast:
AStartPlast (P);
END_STEP

ACTION AStartPlast: #BEGIN_EDIT_BLOCK
IF NOT sv_bPlastEndReached THEN
   fbStart(DeviceId := sv_DeviceId,
        MoveDir := cMoveBwd,
        MoveId := cMovePlast);
ELSE
   //plast not started
   b := WRITE_SV_DIRECT(sv_PlastTimesAct.dActMoveTime, dNull);
   sv_rPlastStartPosition := sv_rScrewPosition;
   b := WRITE_SVREAL_DIRECT(sv_rPlastEndPosition, sv_rPlastStartPosition);
END_IF;

;#END_EDIT_BLOCK END_ACTION (*AStartPlast*)
STEP S_CheckDecAftPlast:
END_STEP

STEP S_DecAftPlast:
AStartDecAftPlast (P);
END_STEP

ACTION AStartDecAftPlast: #BEGIN_EDIT_BLOCK
fbStart(DeviceId := sv_DeviceId,
        MoveDir := cMoveBwd,
        MoveId := cMoveDecompAftPlast);

;#END_EDIT_BLOCK END_ACTION (*AStartDecAftPlast*)
STEP S_Ready:
END_STEP

STEP S_Stop:
AReady (P);
Action17 (P);
AMoveTime (R);
END_STEP

ACTION AReady: #BEGIN_EDIT_BLOCK
fbDebugTrace2(nDeviceState, 'Combined Plast Ready');
sv_bCombinedPlastReady := TRUE;
STOP_PROCESS_ALGORITHM();

;#END_EDIT_BLOCK END_ACTION (*AReady*)
ACTION Action17: #BEGIN_EDIT_BLOCK
//modify pbDeviceReady
sv_DeviceMovements[miIndex].pbDeviceReady := @sv_bDeviceReady;

// sending stopped-Message
evStartedStoppedData.DeviceId := sv_DeviceId;
evStartedStoppedData.MoveId := cMoveCombinedPlast;
evStartedStoppedData.MoveDir := cMoveBwd;
evStartedStoppedData.State := nStopped;
SET_EVENT(evStartedStopped,evStartedStoppedData);

;#END_EDIT_BLOCK END_ACTION (*Action17*)

(* transitions *)
GO_ON_TRANSITION Trans1 (* Trans1 *) FROM S_Init TO S_Start :=  #BEGIN_EDIT_BLOCK
TRUE
;#END_EDIT_BLOCK
END_TRANSITION

GO_ON_TRANSITION TDecBefPlastActivated (* Trans10 *) FROM S_Start TO S_DecBefPlast :=  #BEGIN_EDIT_BLOCK
sv_bActivatedDecompBeforePlast
;#END_EDIT_BLOCK
END_TRANSITION

GO_ON_TRANSITION TDecBefPlastReady (* Trans6 *) FROM S_DecBefPlast TO S_Plast :=  #BEGIN_EDIT_BLOCK
sv_bDeviceReady
;#END_EDIT_BLOCK
END_TRANSITION

GO_ON_TRANSITION TDecBefPlastNotActivated (* Trans29 *) FROM S_Start TO S_Plast :=  #BEGIN_EDIT_BLOCK
NOT sv_bActivatedDecompBeforePlast
;#END_EDIT_BLOCK
END_TRANSITION

GO_ON_TRANSITION TPlastReady (* Trans2 *) FROM S_Plast TO S_CheckDecAftPlast :=  #BEGIN_EDIT_BLOCK
sv_bDeviceReady
;#END_EDIT_BLOCK
END_TRANSITION

GO_ON_TRANSITION TDecAftPlastActivated (* Trans31 *) FROM S_CheckDecAftPlast TO S_DecAftPlast :=  #BEGIN_EDIT_BLOCK
sv_bActivatedDecompAfterPlast
;#END_EDIT_BLOCK
END_TRANSITION

GO_ON_TRANSITION TDecAftPastReady (* Trans6 *) FROM S_DecAftPlast TO S_Ready :=  #BEGIN_EDIT_BLOCK
sv_bDeviceReady
;#END_EDIT_BLOCK
END_TRANSITION

GO_ON_TRANSITION TDecAftPlastNotActivated (* Trans30 *) FROM S_CheckDecAftPlast TO S_Ready :=  #BEGIN_EDIT_BLOCK
NOT sv_bActivatedDecompAfterPlast
;#END_EDIT_BLOCK
END_TRANSITION

GO_ON_TRANSITION TDeviceReady (* Trans28 *) FROM S_Ready TO S_Stop :=  #BEGIN_EDIT_BLOCK
sv_bDeviceReady
;#END_EDIT_BLOCK
END_TRANSITION

TRANSITION Trans11 (* Trans11 *) FROM S_Stop TO S_Start :=  #BEGIN_EDIT_BLOCK
TRUE
;#END_EDIT_BLOCK
END_TRANSITION

(* end IecGraph-Code *)
(* sfc-code *)

(* stand alone actions *)
ACTION AMoveTime: #BEGIN_EDIT_BLOCK
(**************************************** WARNING ********************************************
 *** The KEBA Kemro K2 System including software is not intended for safety control tasks! ***
 ***                       For further information see Comment tab!                        ***
 *********************************************************************************************)

fbMoveTime(IN := TRUE);
b := WRITE_SV_DIRECT(sv_dActPlastDecompTime, fbMoveTime.ET)

;#END_EDIT_BLOCK END_ACTION (*AMoveTime*)

(* exits *)

EXIT_TRANSITION Stop := #BEGIN_EDIT_BLOCK
mbStop
;#END_EDIT_BLOCK
PRIORITY 1 WITH
(* init step *)
INITIAL_STEP Step18:
Action24 (P);
END_STEP

ACTION Action24: #BEGIN_EDIT_BLOCK
mbStop := FALSE;

;#END_EDIT_BLOCK END_ACTION (*Action24*)
STEP S_Ready:
END_STEP

(* steps *)

(* transitions *)
GO_ON_TRANSITION Trans19 (* Trans19 *) FROM Step18 TO S_Ready :=  #BEGIN_EDIT_BLOCK
TRUE
;#END_EDIT_BLOCK
END_TRANSITION

END_TRANSITION
(* end sfc-code *)

END_ALGORITHM

POSTUPDATE_ALGORITHM pPlastProfile ON PU_Task_7 WITH sv_bInitStart,sv_PlastProfVis.Profile,sv_rTargetValueDecBefPlast

#BEGIN_EDIT_BLOCK
(**************************************** WARNING ********************************************
 *** The KEBA Kemro K2 System including software is not intended for safety control tasks! ***
 ***                       For further information see Comment tab!                        ***
 *********************************************************************************************)

IF sv_rTargetValueDecBefPlast < sv_PlastProfVis.Profile.Points[(sv_PlastProfVis.Profile.iNoOfPoints+1)].rStartPos THEN
   sv_CombinedPlastData.Plast.prTargetValue := @sv_PlastProfVis.Profile.Points[(sv_PlastProfVis.Profile.iNoOfPoints+1)].rStartPos;

   //set plast duration to a default value
   //(for displaying in machine sequencer)
   sv_dCalculatedDurationPlast := t#2s;
ELSE
   //decomp before bigger than plast endpos
   sv_CombinedPlastData.Plast.prTargetValue := @sv_rTargetValueDecBefPlast;

   //set plast duration to 0.0s
   sv_dCalculatedDurationPlast := t#0s;
END_IF;

;#END_EDIT_BLOCK END_ALGORITHM

POSTUPDATE_ALGORITHM pDuration ON PU_Task_7 WITH sv_dCalculatedDurationDecompAft,sv_dCalculatedDurationDecompBef,sv_dCalculatedDurationPlast,sv_PlastTimesSet.dSetDelayTime,sv_DecompTimesSet.dSetDelayTime,sv_DecompAftPlastSettings.Mode,sv_DecompBefPlastSettings.Mode

VAR
 dDelayDecompBefore : TIME;
 dDelayDecompAfter : TIME;
 dMoveTime : TIME;
END_VAR
#BEGIN_EDIT_BLOCK
(**************************************** WARNING ********************************************
 *** The KEBA Kemro K2 System including software is not intended for safety control tasks! ***
 ***                       For further information see Comment tab!                        ***
 *********************************************************************************************)

IF sv_DecompBefPlastSettings.Mode <> nNotUsed THEN
   dDelayDecompBefore := sv_DecompTimesSet.dSetDelayTime;
   sv_CombinedPlastData.DecompBefore.pdDelayTime := @sv_DecompTimesSet.dSetDelayTime;
ELSE
   dDelayDecompBefore := t#0s;
   sv_CombinedPlastData.DecompBefore.pdDelayTime := EMPTY;
END_IF;

IF sv_DecompAftPlastSettings.Mode <> nNotUsed THEN
   dDelayDecompAfter := sv_DecompTimesSet.dSetDelayTime;
   sv_CombinedPlastData.DecompAfter.pdDelayTime := @sv_DecompTimesSet.dSetDelayTime;
ELSE
   dDelayDecompAfter := t#0s;
   sv_CombinedPlastData.DecompAfter.pdDelayTime := EMPTY;
END_IF;

IF sv_OperationMode <= nHalfAutomatic THEN
   //in HA and FA the duration of combined plast movement is updated by ODC
   dMoveTime := sv_dCalculatedDurationDecompAft +  sv_dCalculatedDurationDecompBef + sv_dCalculatedDurationPlast;
   sv_dDurationCombinedPlast := dMoveTime + dDelayDecompBefore + dDelayDecompAfter + sv_PlastTimesSet.dSetDelayTime;
END_IF;

;#END_EDIT_BLOCK END_ALGORITHM

POSTUPDATE_ALGORITHM pCompleteDuration ON PU_Task_7 WITH sv_dDurationCombinedPlast

VAR
 fbUpdateProperties : FBUpdateEditorProperties;
END_VAR
#BEGIN_EDIT_BLOCK
(**************************************** WARNING ********************************************
 *** The KEBA Kemro K2 System including software is not intended for safety control tasks! ***
 ***                       For further information see Comment tab!                        ***
 *********************************************************************************************)

fbUpdateProperties();

;#END_EDIT_BLOCK END_ALGORITHM

POSTUPDATE_ALGORITHM pMoveRegisterDone ON PU_Task_7 WITH sv_bMoveRegisterDone

VAR_TEMP
 i : DINT;
END_VAR
#BEGIN_EDIT_BLOCK
(**************************************** WARNING ********************************************
 *** The KEBA Kemro K2 System including software is not intended for safety control tasks! ***
 ***                       For further information see Comment tab!                        ***
 *********************************************************************************************)

//get index of function unit in sv_DeviceMovements - list
FOR i := 1 TO cMaxMoveDevicesRegistered DO
   IF sv_DeviceMovements[i].DeviceId = sv_DeviceId THEN
      miIndex := i;
      EXIT;
   END_IF;
END_FOR;

;#END_EDIT_BLOCK END_ALGORITHM

END_ALGORITHM_BLOCK

#END_OF_IEC_PART

@Puma @IecEditor 6 103 @Pou 25
@@@BEG_Comment@@@
@h    ! WARNING !
@h    The Kemro K2 system (including software) only meets category B according to EN 954-1,
@h    thus it is not intended for usage in safety-relevant control applications in the field
@h    of personal safety (e.g. emergency stop).
@h    To implement potentially necessary safety-relevant control tasks, always use additional
@h    external safety devices that are intended for the particular purpose, and meet the necessary
@h    functional safety.
@h    For further information see EN 954-1 (EN ISO 13849-1) and/or the K2-x00 user manual, chapter
@h    "CE conformity, directives and standards".

ABMoveCombinedPlast is a combination of the following movements:
- decompression before plast
- plast
- decompression after plast

Therefore the movement sv_MoveCombinedPlast is registered

After receiving a start event for the movement with moveId cMoveCombinedPlast this block
coordinates decompression and plast by sending the start events to this movements.

Attention:
To avoid that autocycle continues to early the pbDeviceReady flag is modified.
During this combined movement is active, pbDeviceReady refers to sv_bCombinedPlastReady.
After the movement was stopped or it is finished, pbDeviceReady refers to sv_bDeviceReady again.
@@@END_Comment@@@

@BEG_Contents

@BEG_Func
@RT(17)FuncTreeContainer
1
@Var @RT(9)SET_EVENT @RT(0) @T @T @DERIVED 0 @F @RT(23)KEBA_STANDARD_PROCEDURE @F
@T
@BEG_Attrib
0 @RT(0) @RT(0)
@END_Attrib
1 1 @F @F @F @F

@END_Func

@BEG_Const
@RT(18)ConstTreeContainer
3
@Var @RT(14)cCompInjection @RT(0) @T @F @DT @RT(4)DINT @RT(0) @T @T @BASIC 0 @F
@F @F
@T
@BEG_Attrib
0 @RT(3)104 @RT(19)Component Injection
@END_Attrib
1 1 @F @F @F @F

@Var @RT(19)cMoveDecompBefPlast @RT(0) @T @F @DT @RT(4)DINT @RT(0) @T @T @BASIC 0 @F
@F @F
@T
@BEG_Attrib
0 @RT(2)26 @RT(26)decompression before plast
@END_Attrib
1 1 @F @F @F @F

@Var @RT(18)cMoveCombinedPlast @RT(0) @T @F @DT @RT(4)DINT @RT(0) @T @T @BASIC 0 @F
@F @F
@T
@BEG_Attrib
0 @RT(2)55 @RT(60)combined plast movement (decomp before, plast, decomp after)
@END_Attrib
1 1 @F @F @F @F

@END_Const

@BEG_Export

@BEG_Kind
@ALGORITHM_BLOCK @RT(19)ABMoveCombinedPlast @STRUCTURED_TEXT
@RT(0) @RT(0) @RT(0)
@END_Kind

@BEG_Dcl
@RT(16)DclTreeContainer
38
@Var @RT(20)sv_MoveCombinedPlast @RT(0) @T @T @DERIVED 0 @T @T @DT @RT(10)tsMoveData @RT(0) @T @T @UNKNOWN 0 @F
@F @F
@T
@BEG_Attrib
3 @RT(0) @RT(61)combined plast movement (decomp bef -> plast -> decomp after) @RT(0)
@END_Attrib
1 8 @F @F @F @F

@Var @RT(9)PU_Task_7 @RT(0) @T @T @RENAMED 0 @T @T @DT @RT(4)TASK @RT(0) @T @T @BASIC 0 @F
@F @F
@T
@BEG_Attrib
3 @RT(0) @RT(0) @RT(0)
@END_Attrib
1 7 @F @F @F @F

@Var @RT(9)EV_Task_3 @RT(0) @T @T @RENAMED 0 @T @T @DT @RT(4)TASK @RT(0) @T @T @BASIC 0 @F
@F @F
@T
@BEG_Attrib
3 @RT(0) @RT(0) @RT(0)
@END_Attrib
1 7 @F @F @F @F

@Var @RT(13)sv_bInitStart @RT(0) @T @T @RENAMED 0 @T @T @DT @RT(4)BOOL @RT(0) @T @T @BASIC 0 @F
@F @F
@T
@BEG_Attrib
3 @RT(0) @RT(0) @RT(0)
@END_Attrib
1 8 @F @F @F @F

@Var @RT(6)mbStop @RT(0) @T @F @DT @RT(4)BOOL @RT(0) @T @T @BASIC 0 @F
@F @F
@T
@BEG_Attrib
3 @RT(0) @RT(0) @RT(0)
@END_Attrib
1 0 @F @F @F @F

@Var @RT(7)evStart @RT(0) @T @T @DERIVED 0 @T @T @DT @RT(8)tevStart @RT(0) @T @T @UNKNOWN 0 @F
@F @F
@T
@BEG_Attrib
3 @RT(0) @RT(0) @RT(0)
@END_Attrib
1 7 @F @F @F @F

@Var @RT(6)evStop @RT(0) @T @T @DERIVED 0 @T @T @DT @RT(7)tevStop @RT(0) @T @T @UNKNOWN 0 @F
@F @F
@T
@BEG_Attrib
3 @RT(0) @RT(0) @RT(0)
@END_Attrib
1 7 @F @F @F @F

@Var @RT(11)sv_DeviceId @RT(0) @T @T @DERIVED 0 @T @T @DT @RT(10)tsDeviceId @RT(0) @T @T @UNKNOWN 0 @F
@F @F
@T
@BEG_Attrib
3 @RT(0) @RT(0) @RT(0)
@END_Attrib
1 8 @F @F @F @F

@Var @RT(12)fbDebugTrace @RT(0) @T @T @DERIVED 0 @T @T @DT @RT(12)FBDebugTrace @RT(0) @T @T @UNKNOWN 0 @F
@F @F
@T
@BEG_Attrib
3 @RT(0) @RT(0) @RT(0)
@END_Attrib
1 0 @F @F @F @F

@Var @RT(13)sv_TraceLevel @RT(0) @T @T @DERIVED 0 @T @T @DT @RT(12)tsTraceLevel @RT(0) @T @T @UNKNOWN 0 @F
@F @F
@T
@BEG_Attrib
3 @RT(0) @RT(0) @RT(0)
@END_Attrib
1 8 @F @F @F @F

@Var @RT(15)sv_bDeviceReady @RT(0) @T @F @DT @RT(4)BOOL @RT(0) @T @T @BASIC 0 @F
@F @F
@T
@BEG_Attrib
3 @RT(0) @RT(0) @RT(0)
@END_Attrib
1 8 @F @F @F @F

@Var @RT(18)sv_DeviceMovements @RT(0) @T @T @DERIVED 0 @T @T @DT @RT(19)tDeviceMovementList @RT(0) @T @T @UNKNOWN 0 @F
@F @F
@T
@BEG_Attrib
3 @RT(0) @RT(0) @RT(0)
@END_Attrib
1 8 @F @F @F @F

@Var @RT(22)sv_bCombinedPlastReady @RT(0) @T @F @DT @RT(4)BOOL @RT(0) @T @T @BASIC 0 @F
@F @F
@T
@BEG_Attrib
3 @RT(0) @RT(20)combined plast ready @RT(0)
@END_Attrib
1 8 @F @F @F @F

@Var @RT(16)evStartedStopped @RT(0) @T @T @DERIVED 0 @T @T @DT @RT(17)tevStartedStopped @RT(0) @T @T @UNKNOWN 0 @F
@F @F
@T
@BEG_Attrib
3 @RT(0) @RT(0) @RT(0)
@END_Attrib
1 7 @F @F @F @F

@Var @RT(20)evStartedStoppedData @RT(0) @T @T @DERIVED 0 @T @T @DT @RT(21)tevStartedStoppedData @RT(0) @T @T @UNKNOWN 0 @F
@F @F
@T
@BEG_Attrib
3 @RT(0) @RT(0) @RT(0)
@END_Attrib
1 0 @F @F @F @F

@Var @RT(20)sv_CombinedPlastData @RT(0) @T @T @DERIVED 0 @T @T @DT @RT(19)tsCombinedPlastData @RT(0) @T @T @UNKNOWN 0 @F
@F @F
@T
@BEG_Attrib
3 @RT(0) @RT(66)necessary data for diplaying combined plast movement in odc editor @RT(0)
@END_Attrib
1 8 @F @F @F @F

@Var @RT(15)sv_PlastProfVis @RT(0) @T @T @DERIVED 0 @T @T @DT @RT(21)KAPPL_VisProfilePlast @RT(0) @T @T @UNKNOWN 0 @F
@F @F
@T
@BEG_Attrib
3 @RT(0) @RT(0) @RT(0)
@END_Attrib
1 8 @F @F @F @F

@Var @RT(31)sv_dCalculatedDurationDecompAft @RT(0) @T @T @RENAMED 0 @T @T @DT @RT(4)TIME @RT(0) @T @T @BASIC 0 @F
@F @F
@T
@BEG_Attrib
3 @RT(0) @RT(0) @RT(0)
@END_Attrib
1 8 @F @F @F @F

@Var @RT(31)sv_dCalculatedDurationDecompBef @RT(0) @T @T @RENAMED 0 @T @T @DT @RT(4)TIME @RT(0) @T @T @BASIC 0 @F
@F @F
@T
@BEG_Attrib
3 @RT(0) @RT(0) @RT(0)
@END_Attrib
1 8 @F @F @F @F

@Var @RT(27)sv_dCalculatedDurationPlast @RT(0) @T @T @RENAMED 0 @T @T @DT @RT(4)TIME @RT(0) @T @T @BASIC 0 @F
@F @F
@T
@BEG_Attrib
3 @RT(0) @RT(0) @RT(0)
@END_Attrib
1 8 @F @F @F @F

@Var @RT(25)sv_dDurationCombinedPlast @RT(0) @T @F @DT @RT(4)TIME @RT(0) @T @T @BASIC 0 @F
@F @F
@T
@BEG_Attrib
3 @RT(0) @RT(45)Calculated duration for combined plasticizing @RT(0)
@END_Attrib
1 8 @F @F @F @F

@Var @RT(16)sv_PlastTimesSet @RT(0) @T @T @DERIVED 0 @T @T @DT @RT(10)tsSetTimes @RT(0) @T @T @UNKNOWN 0 @F
@F @F
@T
@BEG_Attrib
3 @RT(0) @RT(0) @RT(0)
@END_Attrib
1 8 @F @F @F @F

@Var @RT(25)sv_DecompAftPlastSettings @RT(0) @T @T @DERIVED 0 @T @T @DT @RT(13)tsDecompParam @RT(0) @T @T @UNKNOWN 0 @F
@F @F
@T
@BEG_Attrib
3 @RT(0) @RT(0) @RT(0)
@END_Attrib
1 8 @F @F @F @F

@Var @RT(25)sv_DecompBefPlastSettings @RT(0) @T @T @DERIVED 0 @T @T @DT @RT(13)tsDecompParam @RT(0) @T @T @UNKNOWN 0 @F
@F @F
@T
@BEG_Attrib
3 @RT(0) @RT(0) @RT(0)
@END_Attrib
1 8 @F @F @F @F

@Var @RT(17)sv_DecompTimesSet @RT(0) @T @T @DERIVED 0 @T @T @DT @RT(10)tsSetTimes @RT(0) @T @T @UNKNOWN 0 @F
@F @F
@T
@BEG_Attrib
3 @RT(0) @RT(0) @RT(0)
@END_Attrib
1 8 @F @F @F @F

@Var @RT(19)sv_bPlastEndReached @RT(0) @T @F @DT @RT(4)BOOL @RT(0) @T @T @BASIC 0 @F
@F @F
@T
@BEG_Attrib
3 @RT(0) @RT(44)flag if plast icizing endposition is reached @RT(0)
@END_Attrib
1 8 @F @F @F @F

@Var @RT(16)sv_OperationMode @RT(0) @T @T @DERIVED 0 @T @T @DT @RT(15)tnOperationMode @RT(0) @T @T @UNKNOWN 0 @F
@F @F
@T
@BEG_Attrib
3 @RT(0) @RT(0) @RT(0)
@END_Attrib
1 8 @F @F @F @F

@Var @RT(26)sv_rTargetValueDecBefPlast @RT(0) @T @F @DT @RT(4)REAL @RT(0) @T @T @BASIC 0 @F
@F @F
@T
@BEG_Attrib
3 @RT(0) @RT(44)target value of decomp before plast (in cmł) @RT(0)
@END_Attrib
1 8 @F @F @F @F

@Var @RT(13)TaskSequencer @RT(0) @T @T @RENAMED 0 @T @T @DT @RT(4)TASK @RT(0) @T @T @BASIC 0 @F
@F @F
@T
@BEG_Attrib
3 @RT(0) @RT(0) @RT(0)
@END_Attrib
1 7 @F @F @F @F

@Var @RT(22)sv_dActPlastDecompTime @RT(0) @T @F @DT @RT(4)TIME @RT(0) @T @T @BASIC 0 @F
@F @F
@T
@BEG_Attrib
3 @RT(0) @RT(36)act time for combined plast movement @RT(0)
@END_Attrib
1 8 @F @F @F @F

@Var @RT(30)sv_bActivatedDecompBeforePlast @RT(0) @T @F @DT @RT(4)BOOL @RT(0) @T @T @BASIC 0 @F
@F @F
@T
@BEG_Attrib
3 @RT(0) @RT(75)indicates if movement decompress should be activated if start event is sent @RT(0)
@END_Attrib
1 8 @F @F @F @F

@Var @RT(29)sv_bActivatedDecompAfterPlast @RT(0) @T @F @DT @RT(4)BOOL @RT(0) @T @T @BASIC 0 @F
@F @F
@T
@BEG_Attrib
3 @RT(0) @RT(75)indicates if movement decompress should be activated if start event is sent @RT(0)
@END_Attrib
1 8 @F @F @F @F

@Var @RT(20)sv_bMoveRegisterDone @RT(0) @T @T @RENAMED 0 @T @T @DT @RT(4)BOOL @RT(0) @T @T @BASIC 0 @F
@F @F
@T
@BEG_Attrib
3 @RT(0) @RT(0) @RT(0)
@END_Attrib
1 8 @F @F @F @F

@Var @RT(7)miIndex @RT(0) @T @F @DT @RT(4)DINT @RT(0) @T @T @BASIC 0 @F
@F @F
@T
@BEG_Attrib
3 @RT(0) @RT(44)index of this FU in sv_DeviceMovement - list @RT(0)
@END_Attrib
1 0 @F @F @F @F

@Var @RT(16)sv_PlastTimesAct @RT(0) @T @T @DERIVED 0 @T @T @DT @RT(10)tsActTimes @RT(0) @T @T @UNKNOWN 0 @F
@F @F
@T
@BEG_Attrib
3 @RT(0) @RT(0) @RT(0)
@END_Attrib
1 8 @F @F @F @F

@Var @RT(22)sv_rPlastStartPosition @RT(0) @T @F @DT @RT(4)REAL @RT(0) @T @T @BASIC 0 @F
@F @F
@T
@BEG_Attrib
3 @RT(0) @RT(33)position at starting plasticizing @RT(0)
@END_Attrib
1 8 @F @F @F @F

@Var @RT(20)sv_rPlastEndPosition @RT(0) @T @F @DT @RT(4)REAL @RT(0) @T @T @BASIC 0 @F
@F @F
@T
@BEG_Attrib
3 @RT(0) @RT(31)position at end of plasticizing @RT(0)
@END_Attrib
1 8 @F @F @F @F

@Var @RT(17)sv_rScrewPosition @RT(0) @T @F @DT @RT(4)REAL @RT(0) @T @T @BASIC 0 @F
@F @F
@T
@BEG_Attrib
3 @RT(0) @RT(30)specific screw position im cmł @RT(0)
@END_Attrib
1 8 @F @F @F @F

@END_Dcl

@END_Export

@BEG_Body

9

@BEG_Export

@BEG_Algo
@ALGORITHM @RT(9)aRegister @STRUCTURED_TEXT
@RT(0) @RT(0) @RT(0) @F @F
@END_Algo

@BEG_Dcl
@RT(16)DclTreeContainer
1
@Var @RT(23)abCombinedPlastRegister @RT(0) @T @T @DERIVED 0 @T @T @DT @RT(18)ABMovementRegister @RT(0) @T @T @UNKNOWN 0 @F
@F @F
@T
@BEG_Attrib
3 @RT(0) @RT(0) @RT(0)
@END_Attrib
1 0 @F @F @F @F

@END_Dcl

@END_Export

@BEG_Export

@BEG_Algo
@POSTUPDATE_ALGORITHM @RT(10)pInitStart @STRUCTURED_TEXT
@RT(0) @RT(13)sv_bInitStart @RT(9)PU_Task_7 @F @F
@END_Algo

@BEG_Dcl
@RT(16)DclTreeContainer
0
@END_Dcl

@END_Export

@BEG_Export

@BEG_Algo
@EVENT_ALGORITHM @RT(8)evaStart @STRUCTURED_TEXT
@RT(0) @RT(7)evStart @RT(9)EV_Task_3 @F @F
@END_Algo

@BEG_Dcl
@RT(16)DclTreeContainer
1
@Var @RT(11)evStartData @RT(0) @T @T @DERIVED 0 @T @T @DT @RT(12)tevStartData @RT(0) @T @T @UNKNOWN 0 @F
@F @F
@T
@BEG_Attrib
3 @RT(0) @RT(0) @RT(0)
@END_Attrib
1 1 @F @F @F @F

@END_Dcl

@END_Export

@BEG_Export

@BEG_Algo
@EVENT_ALGORITHM @RT(7)evaStop @STRUCTURED_TEXT
@RT(0) @RT(6)evStop @RT(9)EV_Task_3 @F @F
@END_Algo

@BEG_Dcl
@RT(16)DclTreeContainer
1
@Var @RT(10)evStopData @RT(0) @T @T @DERIVED 0 @T @T @DT @RT(11)tevStopData @RT(0) @T @T @UNKNOWN 0 @F
@F @F
@T
@BEG_Attrib
3 @RT(0) @RT(0) @RT(0)
@END_Attrib
1 1 @F @F @F @F

@END_Dcl

@END_Export

@BEG_Export

@BEG_Algo
@PROCESS_ALGORITHM @RT(13)paMoveControl @SEQUENTIAL_FLOW_CHART
@RT(0) @RT(0) @RT(16)TaskSequencer(1) @F @F
@END_Algo

@BEG_Dcl
@RT(16)DclTreeContainer
5
@Var @RT(7)fbStart @RT(0) @T @T @DERIVED 0 @T @T @DT @RT(7)FBStart @RT(0) @T @T @UNKNOWN 0 @F
@F @F
@T
@BEG_Attrib
3 @RT(0) @RT(0) @RT(0)
@END_Attrib
1 0 @F @F @F @F

@Var @RT(13)fbDebugTrace2 @RT(0) @T @T @DERIVED 0 @T @T @DT @RT(13)FBDebugTrace2 @RT(0) @T @T @UNKNOWN 0 @F
@F @F
@T
@BEG_Attrib
3 @RT(0) @RT(0) @RT(0)
@END_Attrib
1 0 @F @F @F @F

@Var @RT(10)fbMoveTime @RT(0) @T @T @DERIVED 0 @T @T @DT @RT(3)TON @RT(0) @T @T @UNKNOWN 0 @F
@F @F
@T
@BEG_Attrib
3 @RT(0) @RT(0) @RT(0)
@END_Attrib
1 0 @F @F @F @F

@Var @RT(1)b @RT(0) @T @F @DT @RT(4)BOOL @RT(0) @T @T @BASIC 0 @F
@F @F
@T
@BEG_Attrib
3 @RT(0) @RT(0) @RT(0)
@END_Attrib
1 4 @F @F @F @F

@Var @RT(5)dNull @RT(0) @T @F @DT @RT(4)TIME @RT(0) @T @T @BASIC 0 @F
@F @F
@T
@BEG_Attrib
3 @RT(0) @RT(0) @RT(0)
@END_Attrib
1 0 @F @F @F @F

@END_Dcl

@END_Export

@BEG_Export

@BEG_Algo
@POSTUPDATE_ALGORITHM @RT(13)pPlastProfile @STRUCTURED_TEXT
@RT(0) @RT(64)sv_bInitStart,sv_PlastProfVis.Profile,sv_rTargetValueDecBefPlast @RT(9)PU_Task_7 @F @F
@END_Algo

@BEG_Dcl
@RT(16)DclTreeContainer
0
@END_Dcl

@END_Export

@BEG_Export

@BEG_Algo
@POSTUPDATE_ALGORITHM @RT(9)pDuration @STRUCTURED_TEXT
@RT(0) @RT(216)sv_dCalculatedDurationDecompAft,sv_dCalculatedDurationDecompBef,sv_dCalculatedDurationPlast,sv_PlastTimesSet.dSetDelayTime,sv_DecompTimesSet.dSetDelayTime,sv_DecompAftPlastSettings.Mode,sv_DecompBefPlastSettings.Mode @RT(9)PU_Task_7 @F @F
@END_Algo

@BEG_Dcl
@RT(16)DclTreeContainer
3
@Var @RT(18)dDelayDecompBefore @RT(0) @T @F @DT @RT(4)TIME @RT(0) @T @T @BASIC 0 @F
@F @F
@T
@BEG_Attrib
3 @RT(0) @RT(0) @RT(0)
@END_Attrib
1 0 @F @F @F @F

@Var @RT(17)dDelayDecompAfter @RT(0) @T @F @DT @RT(4)TIME @RT(0) @T @T @BASIC 0 @F
@F @F
@T
@BEG_Attrib
3 @RT(0) @RT(0) @RT(0)
@END_Attrib
1 0 @F @F @F @F

@Var @RT(9)dMoveTime @RT(0) @T @F @DT @RT(4)TIME @RT(0) @T @T @BASIC 0 @F
@F @F
@T
@BEG_Attrib
3 @RT(0) @RT(0) @RT(0)
@END_Attrib
1 0 @F @F @F @F

@END_Dcl

@END_Export

@BEG_Export

@BEG_Algo
@POSTUPDATE_ALGORITHM @RT(17)pCompleteDuration @STRUCTURED_TEXT
@RT(0) @RT(25)sv_dDurationCombinedPlast @RT(9)PU_Task_7 @F @F
@END_Algo

@BEG_Dcl
@RT(16)DclTreeContainer
1
@Var @RT(18)fbUpdateProperties @RT(0) @T @T @DERIVED 0 @T @T @DT @RT(24)FBUpdateEditorProperties @RT(0) @T @T @UNKNOWN 0 @F
@F @F
@T
@BEG_Attrib
3 @RT(0) @RT(0) @RT(0)
@END_Attrib
1 0 @F @F @F @F

@END_Dcl

@END_Export

@BEG_Export

@BEG_Algo
@POSTUPDATE_ALGORITHM @RT(17)pMoveRegisterDone @STRUCTURED_TEXT
@RT(0) @RT(20)sv_bMoveRegisterDone @RT(9)PU_Task_7 @F @F
@END_Algo

@BEG_Dcl
@RT(16)DclTreeContainer
1
@Var @RT(1)i @RT(0) @T @F @DT @RT(4)DINT @RT(0) @T @T @BASIC 0 @F
@F @F
@T
@BEG_Attrib
3 @RT(0) @RT(0) @RT(0)
@END_Attrib
1 4 @F @F @F @F

@END_Dcl

@END_Export

@BEG_Body
@TL(13)
(**************************************** WARNING ********************************************
 *** The KEBA Kemro K2 System including software is not intended for safety control tasks! ***
 ***                       For further information see Comment tab!                        ***
 *********************************************************************************************)

//register inject movement
sv_MoveCombinedPlast.LockGroups[1] := cLockGroupHeatingNozzle;
sv_MoveCombinedPlast.LockGroups[2] := cLockGroupSafetyGateNozzle;
sv_MoveCombinedPlast.LockGroups[3] := cLockGroupSafetyGateMold;
sv_MoveCombinedPlast.sIconPath := CONCAT(GET_MY_FU_NAME(),"\hmi\images\movScrewRotate.gif");

abCombinedPlastRegister.aRegister(@sv_MoveCombinedPlast);

@END_Body

@@@BEG_Comment@@@
@TL(0)

@@@END_Comment@@@

@BEG_Body
@TL(9)
(**************************************** WARNING ********************************************
 *** The KEBA Kemro K2 System including software is not intended for safety control tasks! ***
 ***                       For further information see Comment tab!                        ***
 *********************************************************************************************)

IF sv_bInitStart THEN
   aRegister();
END_IF;

@END_Body

@@@BEG_Comment@@@
@TL(0)

@@@END_Comment@@@

@BEG_Body
@TL(29)
(**************************************** WARNING ********************************************
 *** The KEBA Kemro K2 System including software is not intended for safety control tasks! ***
 ***                       For further information see Comment tab!                        ***
 *********************************************************************************************)

IF evStartData.DeviceId.CompId = sv_DeviceId.CompId AND
   evStartData.DeviceId.IndexId = sv_DeviceId.IndexId  THEN

   IF evStartData.MoveId = cMoveCombinedPlast THEN

      //modify pbDeviceReady
      sv_DeviceMovements[miIndex].pbDeviceReady := @sv_bCombinedPlastReady;

      // sending stopped-Message
      evStartedStoppedData.DeviceId := sv_DeviceId;
      evStartedStoppedData.MoveId := cMoveCombinedPlast;
      evStartedStoppedData.MoveDir := cMoveBwd;
      evStartedStoppedData.State := nStarted;
      SET_EVENT(evStartedStopped,evStartedStoppedData);

      sv_bCombinedPlastReady := FALSE;
      mbStop := FALSE;

      START_PROCESS_ALGORITHM(paMoveControl);
   END_IF;

END_IF;

@END_Body

@@@BEG_Comment@@@
@TL(2)
This Algo receives the evStart event, checks the startconditions and starts paMoveControl.

@@@END_Comment@@@

@BEG_Body
@TL(15)
(**************************************** WARNING ********************************************
 *** The KEBA Kemro K2 System including software is not intended for safety control tasks! ***
 ***                       For further information see Comment tab!                        ***
 *********************************************************************************************)

IF evStopData.DeviceId = sv_DeviceId THEN

    IF sv_TraceLevel.bDeviceState THEN
            fbDebugTrace(sText := 'ABMoveCombinedPlast : evStop received');
    END_IF;

   //stopping movement
   mbStop := TRUE;
END_IF;

@END_Body

@@@BEG_Comment@@@
@TL(1)
Receives the stopevent and signalls paMoveControl to stop the running movement.
@@@END_Comment@@@

@BEG_SfcBody
40 29 31

@BEG_SfcData 2
@StepSeq @RT(4)sseq @F 3
@Step @RT(6)S_Init @F @T @F @F @RT(0) @F
@AcbCont @RT(7)unnamed @F 0

@Trans @RT(6)Trans1 @F @T @F @F @T @F @TL(2)
TRUE

@RT(6)Trans1 @F
@Loop @RT(4)loop @F 2
@StepSeq @RT(3)seq @F 9
@Step @RT(7)S_Start @F @F @F @F @RT(0) @F
@AcbCont @RT(7)unnamed @F 2
@Acb @RT(6)AStart @F @T @RT(1)P @RT(0) @F @F @T @TL(4)
fbDebugTrace2(nDeviceState, 'Combined Plast Started');
fbMoveTime(IN := FALSE,
           PT := t#20d);

@F
@Acb @RT(9)AMoveTime @F @F @RT(1)S @RT(0) @F @F @F @F

@AltBranch @RT(3)alt @F 2
@TransSeq @RT(4)tseq @F 3
@Trans @RT(21)TDecBefPlastActivated @F @T @F @F @T @F @TL(2)
sv_bActivatedDecompBeforePlast

@RT(7)Trans10 @F
@Step @RT(13)S_DecBefPlast @F @F @F @F @RT(0) @F
@AcbCont @RT(7)unnamed @F 1
@Acb @RT(17)AStartDecBefPlast @F @T @RT(1)P @RT(0) @F @F @T @TL(4)
fbStart(DeviceId := sv_DeviceId,
        MoveDir := cMoveBwd,
        MoveId := cMoveDecompBefPlast);

@F

@Trans @RT(17)TDecBefPlastReady @F @T @F @F @T @F @TL(2)
sv_bDeviceReady

@RT(6)Trans6 @F

@TransSeq @RT(4)tseq @F 1
@Trans @RT(24)TDecBefPlastNotActivated @F @T @T @F @T @F @TL(2)
NOT sv_bActivatedDecompBeforePlast

@RT(7)Trans29 @F

@Step @RT(7)S_Plast @F @F @F @F @RT(0) @F
@AcbCont @RT(7)unnamed @F 1
@Acb @RT(11)AStartPlast @F @T @RT(1)P @RT(0) @F @F @T @TL(11)
IF NOT sv_bPlastEndReached THEN
   fbStart(DeviceId := sv_DeviceId,
        MoveDir := cMoveBwd,
        MoveId := cMovePlast);
ELSE
   //plast not started
   b := WRITE_SV_DIRECT(sv_PlastTimesAct.dActMoveTime, dNull);
   sv_rPlastStartPosition := sv_rScrewPosition;
   b := WRITE_SVREAL_DIRECT(sv_rPlastEndPosition, sv_rPlastStartPosition);
END_IF;

@F

@Trans @RT(11)TPlastReady @F @T @F @F @T @F @TL(2)
sv_bDeviceReady

@RT(6)Trans2 @F
@Step @RT(18)S_CheckDecAftPlast @F @F @F @F @RT(0) @F
@AcbCont @RT(7)unnamed @F 0

@AltBranch @RT(3)alt @F 2
@TransSeq @RT(4)tseq @F 3
@Trans @RT(21)TDecAftPlastActivated @F @T @F @F @T @F @TL(2)
sv_bActivatedDecompAfterPlast

@RT(7)Trans31 @F
@Step @RT(13)S_DecAftPlast @F @F @F @F @RT(0) @F
@AcbCont @RT(7)unnamed @F 1
@Acb @RT(17)AStartDecAftPlast @F @T @RT(1)P @RT(0) @F @F @T @TL(4)
fbStart(DeviceId := sv_DeviceId,
        MoveDir := cMoveBwd,
        MoveId := cMoveDecompAftPlast);

@F

@Trans @RT(16)TDecAftPastReady @F @T @F @F @T @F @TL(2)
sv_bDeviceReady

@RT(6)Trans6 @F

@TransSeq @RT(4)tseq @F 1
@Trans @RT(24)TDecAftPlastNotActivated @F @T @T @F @T @F @TL(2)
NOT sv_bActivatedDecompAfterPlast

@RT(7)Trans30 @F

@Step @RT(7)S_Ready @F @F @T @F @RT(0) @F
@AcbCont @RT(7)unnamed @F 0

@Trans @RT(12)TDeviceReady @F @T @F @F @T @F @TL(2)
sv_bDeviceReady

@RT(7)Trans28 @F
@Step @RT(6)S_Stop @F @F @F @F @RT(0) @F
@AcbCont @RT(7)unnamed @F 3
@Acb @RT(6)AReady @F @T @RT(1)P @RT(0) @F @F @T @TL(4)
fbDebugTrace2(nDeviceState, 'Combined Plast Ready');
sv_bCombinedPlastReady := TRUE;
STOP_PROCESS_ALGORITHM();

@F
@Acb @RT(8)Action17 @F @T @RT(1)P @RT(0) @F @F @T @TL(10)
//modify pbDeviceReady
sv_DeviceMovements[miIndex].pbDeviceReady := @sv_bDeviceReady;

// sending stopped-Message
evStartedStoppedData.DeviceId := sv_DeviceId;
evStartedStoppedData.MoveId := cMoveCombinedPlast;
evStartedStoppedData.MoveDir := cMoveBwd;
evStartedStoppedData.State := nStopped;
SET_EVENT(evStartedStopped,evStartedStoppedData);

@F
@Acb @RT(9)AMoveTime @F @F @RT(1)R @RT(0) @F @F @F @F

@Trans @RT(7)Trans11 @F @T @T @T @T @T @TL(2)
TRUE

@RT(7)Trans11 @F

@END_SfcData
@SaActions 1
@SaText @RT(9)AMoveTime 1 @TL(8)
(**************************************** WARNING ********************************************
 *** The KEBA Kemro K2 System including software is not intended for safety control tasks! ***
 ***                       For further information see Comment tab!                        ***
 *********************************************************************************************)

fbMoveTime(IN := TRUE);
b := WRITE_SV_DIRECT(sv_dActPlastDecompTime, fbMoveTime.ET)

@SaTrans 0
@SaExits 1
@SaExit @SaText @RT(4)Stop 1 @TL(2)
mbStop

@RT(6)S_Stop @RT(1)1 @T @F @SaSfc @RT(4)Stop 5 @RT(5)DUMMY
@BEG_SfcData 2
@ExitSeq @RT(4)sseq @F 3
@Step @RT(6)Step18 @F @T @F @F @RT(0) @F
@AcbCont @RT(7)unnamed @F 1
@Acb @RT(8)Action24 @F @T @RT(1)P @RT(0) @F @F @T @TL(2)
mbStop := FALSE;

@F

@Trans @RT(7)Trans19 @F @T @F @F @T @F @TL(2)
TRUE

@RT(7)Trans19 @F
@Goto @RT(7)S_Ready @F @F
@END_SfcData

@END_SfcBody

@@@BEG_Comment@@@
@TL(0)

@@@END_Comment@@@

@BEG_Body
@TL(21)
(**************************************** WARNING ********************************************
 *** The KEBA Kemro K2 System including software is not intended for safety control tasks! ***
 ***                       For further information see Comment tab!                        ***
 *********************************************************************************************)

IF sv_rTargetValueDecBefPlast < sv_PlastProfVis.Profile.Points[(sv_PlastProfVis.Profile.iNoOfPoints+1)].rStartPos THEN
   sv_CombinedPlastData.Plast.prTargetValue := @sv_PlastProfVis.Profile.Points[(sv_PlastProfVis.Profile.iNoOfPoints+1)].rStartPos;

   //set plast duration to a default value
   //(for displaying in machine sequencer)
   sv_dCalculatedDurationPlast := t#2s;
ELSE
   //decomp before bigger than plast endpos
   sv_CombinedPlastData.Plast.prTargetValue := @sv_rTargetValueDecBefPlast;

   //set plast duration to 0.0s
   sv_dCalculatedDurationPlast := t#0s;
END_IF;

@END_Body

@@@BEG_Comment@@@
@TL(0)

@@@END_Comment@@@

@BEG_Body
@TL(27)
(**************************************** WARNING ********************************************
 *** The KEBA Kemro K2 System including software is not intended for safety control tasks! ***
 ***                       For further information see Comment tab!                        ***
 *********************************************************************************************)

IF sv_DecompBefPlastSettings.Mode <> nNotUsed THEN
   dDelayDecompBefore := sv_DecompTimesSet.dSetDelayTime;
   sv_CombinedPlastData.DecompBefore.pdDelayTime := @sv_DecompTimesSet.dSetDelayTime;
ELSE
   dDelayDecompBefore := t#0s;
   sv_CombinedPlastData.DecompBefore.pdDelayTime := EMPTY;
END_IF;

IF sv_DecompAftPlastSettings.Mode <> nNotUsed THEN
   dDelayDecompAfter := sv_DecompTimesSet.dSetDelayTime;
   sv_CombinedPlastData.DecompAfter.pdDelayTime := @sv_DecompTimesSet.dSetDelayTime;
ELSE
   dDelayDecompAfter := t#0s;
   sv_CombinedPlastData.DecompAfter.pdDelayTime := EMPTY;
END_IF;

IF sv_OperationMode <= nHalfAutomatic THEN
   //in HA and FA the duration of combined plast movement is updated by ODC
   dMoveTime := sv_dCalculatedDurationDecompAft +  sv_dCalculatedDurationDecompBef + sv_dCalculatedDurationPlast;
   sv_dDurationCombinedPlast := dMoveTime + dDelayDecompBefore + dDelayDecompAfter + sv_PlastTimesSet.dSetDelayTime;
END_IF;

@END_Body

@@@BEG_Comment@@@
@TL(0)

@@@END_Comment@@@

@BEG_Body
@TL(7)
(**************************************** WARNING ********************************************
 *** The KEBA Kemro K2 System including software is not intended for safety control tasks! ***
 ***                       For further information see Comment tab!                        ***
 *********************************************************************************************)

fbUpdateProperties();

@END_Body

@@@BEG_Comment@@@
@TL(0)

@@@END_Comment@@@

@BEG_Body
@TL(13)
(**************************************** WARNING ********************************************
 *** The KEBA Kemro K2 System including software is not intended for safety control tasks! ***
 ***                       For further information see Comment tab!                        ***
 *********************************************************************************************)

//get index of function unit in sv_DeviceMovements - list
FOR i := 1 TO cMaxMoveDevicesRegistered DO
   IF sv_DeviceMovements[i].DeviceId = sv_DeviceId THEN
      miIndex := i;
      EXIT;
   END_IF;
END_FOR;

@END_Body

@@@BEG_Comment@@@
@TL(0)

@@@END_Comment@@@
@END_Body

@END_Contents
